DATA_BLOCK "DB_Alarms"   // DB44
{ S7_Optimized_Access := 'FALSE' }
AUTHOR : Heaten
VERSION : 0.1
// stored: AutoNumber true, DBAccessibleFromOPCUA true, DBAccessibleFromWebserver true, IsOnlyStoredInLoadMemory false, IsWriteProtectedInAS false
   VAR RETAIN
      bAckAll : Bool := FALSE;   // Global alarm acknowledge
      bCommonAlarm : Bool := FALSE;   // Global common alarm
      bCriticalAlarm : Bool := FALSE;   // Global critical alarm
      "0001_WatchdogTimeoutOB1" { S7_SetPoint := 'True'} : "stEvent";
      "0003_InitCurrentSettingsFailed" { S7_SetPoint := 'True'} : "stEvent";
      "1001_ConnectionToWinCClost" { S7_SetPoint := 'True'} : "stEvent";
      "1002_EmergencyStopActive" { S7_SetPoint := 'True'} : "stEvent";
      "1003_EmergencyStopResetFailed" { S7_SetPoint := 'True'} : "stEvent";
      "1004_HBL_PS_500_X2" { S7_SetPoint := 'True'} : "stEvent";
      "1101_HBL_SC_01_CommError" { S7_SetPoint := 'True'} : "stDigitalAlarm";
      "1102_HBL_SC_02_CommError" { S7_SetPoint := 'True'} : "stDigitalAlarm";
      "1103_HBL_SC_03_CommError" { S7_SetPoint := 'True'} : "stDigitalAlarm";
      "1110_HBL_SC_10_CommError" { S7_SetPoint := 'True'} : "stDigitalAlarm";
      "1121_HBL_SC_01_Tripped" { S7_SetPoint := 'True'} : "stDigitalAlarm";
      "1122_HBL_SC_02_Tripped" { S7_SetPoint := 'True'} : "stDigitalAlarm";
      "1123_HBL_SC_03_Tripped" { S7_SetPoint := 'True'} : "stDigitalAlarm";
      "1130_HBL_SC_10_Tripped" { S7_SetPoint := 'True'} : "stDigitalAlarm";
      "1140_HBL_SC_01_RunFailure" { S7_SetPoint := 'True'} : "stDigitalAlarm";
      "1142_HBL_SC_02_RunFailure" { S7_SetPoint := 'True'} : "stDigitalAlarm";
      "1143_HBL_SC_03_RunFailure" { S7_SetPoint := 'True'} : "stDigitalAlarm";
      "1150_HBL_SC_10_RunFailure" { S7_SetPoint := 'True'} : "stDigitalAlarm";
      "1201_HBL_PT_517_Fault" { S7_SetPoint := 'True'} : "stEvent";
      "1202_HBL_PT_612_Fault" { S7_SetPoint := 'True'} : "stEvent";
      "1203_HBL_PT_519_Fault" { S7_SetPoint := 'True'} : "stEvent";
      "1204_HBL_PT_544_Fault" { S7_SetPoint := 'True'} : "stEvent";
      "1205_HBL_TT_516_Fault" { S7_SetPoint := 'True'} : "stEvent";
      "1206_HBL_TT_611_Fault" { S7_SetPoint := 'True'} : "stEvent";
      "1207_HBL_TT_901_Fault" { S7_SetPoint := 'True'} : "stEvent";
      "1208_HBL_TT_518_Fault" { S7_SetPoint := 'True'} : "stEvent";
      "1209_HBL_HCV_576_A1_Fault" { S7_SetPoint := 'True'} : "stEvent";
      "1210_HBL_TT_573_Fault" { S7_SetPoint := 'True'} : "stEvent";
      "1212_HBL_TT_543_Fault" { S7_SetPoint := 'True'} : "stEvent";
      "1213_HBL_TT_546_Fault" { S7_SetPoint := 'True'} : "stEvent";
      "1214_HBL_TT_542_Fault" { S7_SetPoint := 'True'} : "stEvent";
      "1215_HBL_TT_571_Fault" { S7_SetPoint := 'True'} : "stEvent";
      "1216_HBL_TT_16_Fault" { S7_SetPoint := 'True'} : "stEvent";
      "1217_HBL_TT_17_Fault" { S7_SetPoint := 'True'} : "stEvent";
      "1218_HBL_TT_18_Fault" { S7_SetPoint := 'True'} : "stEvent";
      "1220_HBL_PT_960_Fault" { S7_SetPoint := 'True'} : "stEvent";
      "1221_HBL_PT_05_Fault" { S7_SetPoint := 'True'} : "stEvent";
      "1223_HBL_TT_03_Fault" { S7_SetPoint := 'True'} : "stEvent";
      "1224_HBL_TT_23_Fault" { S7_SetPoint := 'True'} : "stEvent";
      "1225_HBL_TT_24_Fault" { S7_SetPoint := 'True'} : "stEvent";
      "1226_HBL_TT_25_Fault" { S7_SetPoint := 'True'} : "stEvent";
      "1227_HBL_LT_610_Fault" { S7_SetPoint := 'True'} : "stEvent";
      "1228_HBL_TT_21_Fault" { S7_SetPoint := 'True'} : "stEvent";
      "1229_HBL_TT_22_Fault" { S7_SetPoint := 'True'} : "stEvent";
      "1230_HBL_LT_02_Fault" { S7_SetPoint := 'True'} : "stEvent";   // Deprecated
      "1231_HBL_HCV_578_A1_Fault" { S7_SetPoint := 'True'} : "stEvent";
      "1232_HBL_PT_503_Fault" { S7_SetPoint := 'True'} : "stEvent";
      "1233_HBL_TT_20_Fault" { S7_SetPoint := 'True'} : "stDigitalAlarm";
      "1234_HBL_PT_14_Fault" { S7_SetPoint := 'True'} : "stEvent";   // Deprecated
      "1235_HBL_PT_18_Fault" { S7_SetPoint := 'True'} : "stEvent";   // Deprecated
      "1236_HBL_PT_19_Fault" { S7_SetPoint := 'True'} : "stEvent";   // Deprecated
      "1237_HBL_PT_25_Fault" { S7_SetPoint := 'True'} : "stEvent";   // Deprecated
      "1238_HBL_TT_31_Fault" { S7_SetPoint := 'True'} : "stEvent";   // Deprecated
      "1239_HBL_TT_33_Fault" { S7_SetPoint := 'True'} : "stEvent";   // Deprecated
      "1240_HBL_TT_35_Fault" { S7_SetPoint := 'True'} : "stEvent";   // Deprecated
      "1241_HBL_HCV_576_Fault" { S7_SetPoint := 'True'} : "stEvent";
      "1242_HBL_HCV_578_Fault" { S7_SetPoint := 'True'} : "stEvent";
      "1243_HBL_PT_902_Fault" { S7_SetPoint := 'True'} : "stEvent";
      "1244_HBL_PT_572_Fault" { S7_SetPoint := 'True'} : "stEvent";
      "1245_HBL_PT_09_Fault" { S7_SetPoint := 'True'} : "stEvent";   // Deprecated
      "1246_HBL_PT_547_Fault" { S7_SetPoint := 'True'} : "stEvent";
      "1247_HBL_PT_541_Fault" { S7_SetPoint := 'True'} : "stEvent";
      "1248_HBL_PT_531_Fault" { S7_SetPoint := 'True'} : "stEvent";
      "1249_HBL_PT_701_Fault" { S7_SetPoint := 'True'} : "stEvent";
      "1251_HBL_PT_534_Fault" { S7_SetPoint := 'True'} : "stEvent";
      "1252_HBL_TT_540_Fault" { S7_SetPoint := 'True'} : "stEvent";
      "1253_HBL_TT_530_Fault" { S7_SetPoint := 'True'} : "stEvent";
      "1254_HBL_TT_533_Fault" { S7_SetPoint := 'True'} : "stEvent";
      "1255_HBL_CT_01_Fault" { S7_SetPoint := 'True'} : "stEvent";
      "1256_HBL_CT_615_Fault" { S7_SetPoint := 'True'} : "stEvent";
      "1257_HBL_CT_03_Fault" { S7_SetPoint := 'True'} : "stEvent";
      "1258_HBL_TT_26_Fault" { S7_SetPoint := 'True'} : "stEvent";
      "1259_HBL_TT_27_Fault" { S7_SetPoint := 'True'} : "stEvent";
      "1260_HBL_FT_520_Fault" { S7_SetPoint := 'True'} : "stEvent";
      "1262_HBL_TT_504_Fault" { S7_SetPoint := 'True'} : "stEvent";
      "1263_HBL_TT_34_Fault" { S7_SetPoint := 'True'} : "stEvent";
      "1264_HBL_PT_961_Fault" { S7_SetPoint := 'True'} : "stEvent";
      "1265_HBL_TT_502_Fault" { S7_SetPoint := 'True'} : "stEvent";
      "1266_HBL_LT_510_Fault" { S7_SetPoint := 'True'} : "stEvent";
      "1267_HBL_PT_511_Fault" { S7_SetPoint := 'True'} : "stEvent";
      "1268_HBL_TT_512_Fault" { S7_SetPoint := 'True'} : "stEvent";
      "1269_HBL_TT_532_Fault" { S7_SetPoint := 'True'} : "stEvent";
      "1270_HBL_AT_535_Fault" { S7_SetPoint := 'True'} : "stEvent";
      "1271_HBL_AT_545_Fault" { S7_SetPoint := 'True'} : "stEvent";
      "1272_HBL_PT_635_Fault" { S7_SetPoint := 'True'} : "stEvent";
      "1273_HBL_PT_636_Fault" { S7_SetPoint := 'True'} : "stEvent";
      "1274_HBL_LT_650_Fault" { S7_SetPoint := 'True'} : "stEvent";
      "1275_HBL_PT_651_Fault" { S7_SetPoint := 'True'} : "stEvent";
      "1276_HBL_PT_702_Fault" { S7_SetPoint := 'True'} : "stEvent";
      "1277_HBL_HCV_514_Fault" { S7_SetPoint := 'True'} : "stEvent";
      "1278_HBL_HCV_514_A1_Fault" { S7_SetPoint := 'True'} : "stEvent";
      "1279_HBL_HCV_515_Fault" { S7_SetPoint := 'True'} : "stEvent";
      "1280_HBL_HCV_515_A1_Fault" { S7_SetPoint := 'True'} : "stEvent";
      "1281_HBL_HCV_548_Fault" { S7_SetPoint := 'True'} : "stEvent";
      "1282_HBL_HCV_548_A1_Fault" { S7_SetPoint := 'True'} : "stEvent";
      "1283_HBL_HCV_575_Fault" { S7_SetPoint := 'True'} : "stEvent";
      "1284_HBL_HCV_575_A1_Fault" { S7_SetPoint := 'True'} : "stEvent";
      "1285_HBL_HCV_577_Fault" { S7_SetPoint := 'True'} : "stEvent";
      "1286_HBL_HCV_577_A1_Fault" { S7_SetPoint := 'True'} : "stEvent";
      "1287_HBL_HCV_579_Fault" { S7_SetPoint := 'True'} : "stEvent";
      "1288_HBL_HCV_579_A1_Fault" { S7_SetPoint := 'True'} : "stEvent";
      "1289_HBL_HCV_616_Fault" { S7_SetPoint := 'True'} : "stEvent";
      "1290_HBL_HCV_616_A1_Fault" { S7_SetPoint := 'True'} : "stEvent";
      "1291_HBL_HCV_700_Fault" { S7_SetPoint := 'True'} : "stEvent";
      "1292_HBL_HCV_700_A1_Fault" { S7_SetPoint := 'True'} : "stEvent";
      "1293_HBL_PT_618_Fault" { S7_SetPoint := 'True'} : "stEvent";
      "1294_HBL_LS_632_Fault" { S7_SetPoint := 'True'} : "stDigitalAlarm";
      "1295_HBL_LS_633_Fault" { S7_SetPoint := 'True'} : "stDigitalAlarm";
      "2018_HBL_PT_05_High" { S7_SetPoint := 'True'} : "stLimitAlarm";
      "2028_HBL_PT_17_Low" { S7_SetPoint := 'True'} : "stLimitAlarm";
      "2058_HBL_TT_03_Low" { S7_SetPoint := 'True'} : "stLimitAlarm";
      "2100_HBL_TT_03_High" { S7_SetPoint := 'True'} : "stLimitAlarm";
      "2101_HBL_TT_901_High" { S7_SetPoint := 'True'} : "stLimitAlarm";
      "2102_HBL_PT_503_High" { S7_SetPoint := 'True'} : "stLimitAlarm";
      "2103_HBL_TT_518_High" { S7_SetPoint := 'True'} : "stLimitAlarm";
      "2105_HBL_TT_546_High" { S7_SetPoint := 'True'} : "stLimitAlarm";
      "2106_HBL_TT_17_High" { S7_SetPoint := 'True'} : "stLimitAlarm";
      "2107_HBL_TT_16_High" { S7_SetPoint := 'True'} : "stLimitAlarm";
      "2108_HBL_TT_18_High" { S7_SetPoint := 'True'} : "stLimitAlarm";
      "2109_HBL_TT_20_High" { S7_SetPoint := 'True'} : "stLimitAlarm";
      "2110_HBL_TT_21_High" { S7_SetPoint := 'True'} : "stLimitAlarm";
      "2111_HBL_TT_22_High" { S7_SetPoint := 'True'} : "stLimitAlarm";
      "2112_HBL_LT_02_High" { S7_SetPoint := 'True'} : "stLimitAlarm";   // Deprecated
      "2113_HBL_CT_01_High" { S7_SetPoint := 'True'} : "stLimitAlarm";
      "2114_HBL_CT_615_High" { S7_SetPoint := 'True'} : "stLimitAlarm";
      "2115_HBL_PT_17_LowLow" { S7_SetPoint := 'True'} : "stLimitAlarm";
      "2116_HBL_PT_503_HighHigh" { S7_SetPoint := 'True'} : "stLimitAlarm";
      "2117_HBL_TT_542_Low" { S7_SetPoint := 'True'} : "stLimitAlarm";
      "2301_HeatSourceTempDropCritical" { S7_SetPoint := 'True'} : "stLimitAlarm";
      "2302_HeatSourceTempRiseCritical" { S7_SetPoint := 'True'} : "stLimitAlarm";
      "2303_SuperheatCompressor_High" { S7_SetPoint := 'True'} : "stLimitAlarm";
      "2304_SuperheatCompressor_Low" { S7_SetPoint := 'True'} : "stLimitAlarm";
      "2305_OilFilterDeltaP_High" { S7_SetPoint := 'True'} : "stLimitAlarm";
      "2306_OilFilterDeltaP_HighHigh" { S7_SetPoint := 'True'} : "stLimitAlarm";
      "2307_EvaporatorDischargePressureMeanValue" { S7_SetPoint := 'True'} : "stEvent";
      "2308_EvaporatorDischargePressureHigh" { S7_SetPoint := 'True'} : "stLimitAlarm";
      "2309_OilSeparatorStage1High" { S7_SetPoint := 'True'} : "stDigitalAlarm";
      "3020_SuperheatControlRegulatorFault" { S7_SetPoint := 'True'} : "stEvent";
      "3030_PinchControlRegulatorfault" { S7_SetPoint := 'True'} : "stEvent";
      "3400_HydrolockProtectionActive" { S7_SetPoint := 'True'} : "stEvent";
      "3401_DripPanLevelHigh" { S7_SetPoint := 'True'} : "stDigitalAlarm";
      "5000_OilHeatingActivationFailure" { S7_SetPoint := 'True'} : "stDigitalAlarm";
      "5001_OilHeatingDeactivationFailure" { S7_SetPoint := 'True'} : "stDigitalAlarm";
      "5200_CPC_LT_870_Fault" { S7_SetPoint := 'True'} : "stEvent";
      "5201_CPC_TT_871_Fault" { S7_SetPoint := 'True'} : "stEvent";
      "5202_CPC_PT_872_Fault" { S7_SetPoint := 'True'} : "stEvent";
      "5203_CPC_SC_01_CommError" { S7_SetPoint := 'True'} : "stDigitalAlarm";   // Deprecated
      "5204_CPC_SC_01_Tripped" { S7_SetPoint := 'True'} : "stDigitalAlarm";   // Deprecated
      "5205_CPC_LT_870_High" { S7_SetPoint := 'True'} : "stLimitAlarm";
      "5206_CPC_PT_862_Fault" { S7_SetPoint := 'True'} : "stEvent";
      "5250_SSC_TT_01_Fault" { S7_SetPoint := 'True'} : "stEvent";
      "5251_SSC_TT_02_Fault" { S7_SetPoint := 'True'} : "stEvent";
      "5252_SSC_TT_03_Fault" { S7_SetPoint := 'True'} : "stEvent";
      "5253_SSC_TT_04_Fault" { S7_SetPoint := 'True'} : "stEvent";
      "5254_SSC_PIT_01_Fault" { S7_SetPoint := 'True'} : "stEvent";
      "5255_SSC_PDT_01_Fault" { S7_SetPoint := 'True'} : "stEvent";
      "5256_SSC_LT_01_Fault" { S7_SetPoint := 'True'} : "stEvent";
      "5257_SSC_LT_01_Low" { S7_SetPoint := 'True'} : "stLimitAlarm";
      "5258_SSC_PDT_01_High" { S7_SetPoint := 'True'} : "stLimitAlarm";
      "5259_SSC_TT_02_High" { S7_SetPoint := 'True'} : "stLimitAlarm";
      "5260_SSC_TT_03_Low" { S7_SetPoint := 'True'} : "stLimitAlarm";
      "5261_SSC_PIT_01_Low" { S7_SetPoint := 'True'} : "stLimitAlarm";
      "5262_DeltaT_ShaftSealHigh" { S7_SetPoint := 'True'} : "stLimitAlarm";
      "5263_SSC_PIT_01_High" { S7_SetPoint := 'True'} : "stLimitAlarm";
      "5268_ShaftSealSystemShutdown" { S7_SetPoint := 'True'} : "stDigitalAlarm";
      "9023_HBL_HCV_576_Deviation" { S7_SetPoint := 'True'} : "stDeviationAlarm";
      "9024_HBL_HCV_578_Deviation" { S7_SetPoint := 'True'} : "stDeviationAlarm";
      "9025_HBL_HCV_577_Deviation" { S7_SetPoint := 'True'} : "stDeviationAlarm";
      "9026_HBL_HCV_579_Deviation" { S7_SetPoint := 'True'} : "stDeviationAlarm";
      "9027_HBL_HCV_575_Deviation" { S7_SetPoint := 'True'} : "stDeviationAlarm";
      "9028_HBL_HCV_616_Deviation" { S7_SetPoint := 'True'} : "stDeviationAlarm";
      "9029_HBL_HCV_700_Deviation" { S7_SetPoint := 'True'} : "stDeviationAlarm";
      "9030_HBL_HCV_514_Deviation" { S7_SetPoint := 'True'} : "stDeviationAlarm";
      "9031_HBL_HCV_548_Deviation" { S7_SetPoint := 'True'} : "stDeviationAlarm";
   END_VAR
BEGIN
   "0001_WatchdogTimeoutOB1".bEnable := true;
   "0003_InitCurrentSettingsFailed".bEnable := TRUE;
   "1001_ConnectionToWinCClost".bEnable := TRUE;
   "1002_EmergencyStopActive".bEnable := TRUE;
   "1003_EmergencyStopResetFailed".bEnable := TRUE;
   "1101_HBL_SC_01_CommError".bEnable := true;
   "1101_HBL_SC_01_CommError".bInput := FALSE;
   "1101_HBL_SC_01_CommError".tActivationDelay := T#1S;
   "1102_HBL_SC_02_CommError".bEnable := true;
   "1102_HBL_SC_02_CommError".tActivationDelay := T#1s;
   "1103_HBL_SC_03_CommError".bEnable := true;
   "1103_HBL_SC_03_CommError".tActivationDelay := T#1s;
   "1110_HBL_SC_10_CommError".bEnable := TRUE;
   "1110_HBL_SC_10_CommError".bInput := FALSE;
   "1110_HBL_SC_10_CommError".tActivationDelay := T#5s;
   "1121_HBL_SC_01_Tripped".bEnable := TRUE;
   "1121_HBL_SC_01_Tripped".bInput := FALSE;
   "1121_HBL_SC_01_Tripped".tActivationDelay := T#0MS;
   "1122_HBL_SC_02_Tripped".bEnable := true;
   "1122_HBL_SC_02_Tripped".tActivationDelay := T#0s;
   "1123_HBL_SC_03_Tripped".bEnable := true;
   "1130_HBL_SC_10_Tripped".bEnable := TRUE;
   "1130_HBL_SC_10_Tripped".bInput := FALSE;
   "1130_HBL_SC_10_Tripped".tActivationDelay := T#3s;
   "1140_HBL_SC_01_RunFailure".bEnable := TRUE;
   "1140_HBL_SC_01_RunFailure".bInput := FALSE;
   "1140_HBL_SC_01_RunFailure".tActivationDelay := T#0MS;
   "1142_HBL_SC_02_RunFailure".bEnable := true;
   "1142_HBL_SC_02_RunFailure".tActivationDelay := T#3s;
   "1143_HBL_SC_03_RunFailure".bEnable := true;
   "1143_HBL_SC_03_RunFailure".tActivationDelay := T#3s;
   "1150_HBL_SC_10_RunFailure".bEnable := TRUE;
   "1150_HBL_SC_10_RunFailure".bInput := FALSE;
   "1150_HBL_SC_10_RunFailure".tActivationDelay := T#3s;
   "1201_HBL_PT_517_Fault".bEnable := true;
   "1202_HBL_PT_612_Fault".bEnable := true;
   "1203_HBL_PT_519_Fault".bEnable := true;
   "1204_HBL_PT_544_Fault".bEnable := true;
   "1205_HBL_TT_516_Fault".bEnable := true;
   "1206_HBL_TT_611_Fault".bEnable := true;
   "1207_HBL_TT_901_Fault".bEnable := true;
   "1208_HBL_TT_518_Fault".bEnable := true;
   "1209_HBL_HCV_576_A1_Fault".bEnable := true;
   "1210_HBL_TT_573_Fault".bEnable := true;
   "1212_HBL_TT_543_Fault".bEnable := true;
   "1213_HBL_TT_546_Fault".bEnable := true;
   "1214_HBL_TT_542_Fault".bEnable := true;
   "1215_HBL_TT_571_Fault".bEnable := true;
   "1216_HBL_TT_16_Fault".bEnable := true;
   "1217_HBL_TT_17_Fault".bEnable := true;
   "1218_HBL_TT_18_Fault".bEnable := true;
   "1220_HBL_PT_960_Fault".bEnable := true;
   "1221_HBL_PT_05_Fault".bEnable := true;
   "1223_HBL_TT_03_Fault".bEnable := true;
   "1224_HBL_TT_23_Fault".bEnable := true;
   "1225_HBL_TT_24_Fault".bEnable := true;
   "1226_HBL_TT_25_Fault".bEnable := true;
   "1227_HBL_LT_610_Fault".bEnable := true;
   "1228_HBL_TT_21_Fault".bEnable := true;
   "1229_HBL_TT_22_Fault".bEnable := true;
   "1230_HBL_LT_02_Fault".bEnable := false;
   "1231_HBL_HCV_578_A1_Fault".bEnable := true;
   "1232_HBL_PT_503_Fault".bEnable := true;
   "1233_HBL_TT_20_Fault".bEnable := TRUE;
   "1233_HBL_TT_20_Fault".tActivationDelay := T#5S;
   "1234_HBL_PT_14_Fault".bEnable := true;
   "1235_HBL_PT_18_Fault".bEnable := true;
   "1236_HBL_PT_19_Fault".bEnable := true;
   "1237_HBL_PT_25_Fault".bEnable := false;
   "1238_HBL_TT_31_Fault".bEnable := true;
   "1239_HBL_TT_33_Fault".bEnable := true;
   "1240_HBL_TT_35_Fault".bEnable := true;
   "1241_HBL_HCV_576_Fault".bEnable := true;
   "1242_HBL_HCV_578_Fault".bEnable := true;
   "1243_HBL_PT_902_Fault".bEnable := true;
   "1244_HBL_PT_572_Fault".bEnable := true;
   "1245_HBL_PT_09_Fault".bEnable := true;
   "1246_HBL_PT_547_Fault".bEnable := true;
   "1247_HBL_PT_541_Fault".bEnable := true;
   "1248_HBL_PT_531_Fault".bEnable := true;
   "1249_HBL_PT_701_Fault".bEnable := true;
   "1251_HBL_PT_534_Fault".bEnable := true;
   "1252_HBL_TT_540_Fault".bEnable := true;
   "1253_HBL_TT_530_Fault".bEnable := true;
   "1254_HBL_TT_533_Fault".bEnable := true;
   "1255_HBL_CT_01_Fault".bEnable := true;
   "1256_HBL_CT_615_Fault".bEnable := true;
   "1258_HBL_TT_26_Fault".bEnable := true;
   "1259_HBL_TT_27_Fault".bEnable := true;
   "1260_HBL_FT_520_Fault".bEnable := true;
   "1262_HBL_TT_504_Fault".bEnable := true;
   "1263_HBL_TT_34_Fault".bEnable := true;
   "1264_HBL_PT_961_Fault".bEnable := true;
   "1265_HBL_TT_502_Fault".bEnable := true;
   "1266_HBL_LT_510_Fault".bEnable := true;
   "1267_HBL_PT_511_Fault".bEnable := true;
   "1268_HBL_TT_512_Fault".bEnable := true;
   "1269_HBL_TT_532_Fault".bEnable := true;
   "1270_HBL_AT_535_Fault".bEnable := true;
   "1271_HBL_AT_545_Fault".bEnable := true;
   "1272_HBL_PT_635_Fault".bEnable := true;
   "1273_HBL_PT_636_Fault".bEnable := true;
   "1274_HBL_LT_650_Fault".bEnable := true;
   "1275_HBL_PT_651_Fault".bEnable := true;
   "1276_HBL_PT_702_Fault".bEnable := true;
   "1283_HBL_HCV_575_Fault".bEnable := true;
   "1284_HBL_HCV_575_A1_Fault".bEnable := true;
   "1285_HBL_HCV_577_Fault".bEnable := true;
   "1286_HBL_HCV_577_A1_Fault".bEnable := true;
   "1287_HBL_HCV_579_Fault".bEnable := true;
   "1288_HBL_HCV_579_A1_Fault".bEnable := true;
   "1289_HBL_HCV_616_Fault".bEnable := true;
   "1290_HBL_HCV_616_A1_Fault".bEnable := true;
   "1291_HBL_HCV_700_Fault".bEnable := true;
   "1292_HBL_HCV_700_A1_Fault".bEnable := true;
   "1293_HBL_PT_618_Fault".bEnable := true;
   "1294_HBL_LS_632_Fault".tActivationDelay := t#5S;
   "2018_HBL_PT_05_High".bEnable := true;
   "2018_HBL_PT_05_High".fLimit := 1600.0;
   "2018_HBL_PT_05_High".fHysteresis := 0.0;
   "2018_HBL_PT_05_High".tActivationDelay := T#0MS;
   "2028_HBL_PT_17_Low".bEnable := true;
   "2028_HBL_PT_17_Low".fLimit := 30.0;
   "2028_HBL_PT_17_Low".fHysteresis := 0.0;
   "2028_HBL_PT_17_Low".tActivationDelay := T#30s;
   "2058_HBL_TT_03_Low".bEnable := true;
   "2058_HBL_TT_03_Low".fLimit := 0.0;
   "2058_HBL_TT_03_Low".fHysteresis := 1.0;
   "2058_HBL_TT_03_Low".tActivationDelay := T#180s;
   "2100_HBL_TT_03_High".bEnable := true;
   "2100_HBL_TT_03_High".tActivationDelay := T#0MS;
   "2101_HBL_TT_901_High".bEnable := true;
   "2101_HBL_TT_901_High".fHysteresis := 5.0;
   "2101_HBL_TT_901_High".tActivationDelay := T#5s;
   "2102_HBL_PT_503_High".bEnable := true;
   "2102_HBL_PT_503_High".tActivationDelay := T#1s;
   "2103_HBL_TT_518_High".bEnable := true;
   "2103_HBL_TT_518_High".tActivationDelay := T#1s;
   "2105_HBL_TT_546_High".bEnable := true;
   "2106_HBL_TT_17_High".bEnable := true;
   "2106_HBL_TT_17_High".tActivationDelay := T#10s;
   "2107_HBL_TT_16_High".bEnable := true;
   "2107_HBL_TT_16_High".tActivationDelay := T#10s;
   "2108_HBL_TT_18_High".bEnable := true;
   "2108_HBL_TT_18_High".tActivationDelay := T#10s;
   "2109_HBL_TT_20_High".bEnable := true;
   "2109_HBL_TT_20_High".tActivationDelay := T#0s;
   "2110_HBL_TT_21_High".bEnable := true;
   "2110_HBL_TT_21_High".fHysteresis := 5.0;
   "2110_HBL_TT_21_High".tActivationDelay := T#10s;
   "2111_HBL_TT_22_High".bEnable := true;
   "2111_HBL_TT_22_High".fHysteresis := 5.0;
   "2111_HBL_TT_22_High".tActivationDelay := T#10s;
   "2112_HBL_LT_02_High".bEnable := true;
   "2112_HBL_LT_02_High".tActivationDelay := T#5s;
   "2113_HBL_CT_01_High".bEnable := true;
   "2113_HBL_CT_01_High".fHysteresis := 50.0;
   "2114_HBL_CT_615_High".bEnable := true;
   "2114_HBL_CT_615_High".fHysteresis := 50.0;
   "2115_HBL_PT_17_LowLow".bEnable := true;
   // "2115_HBL_PT_17_LowLow".fLimit : Dynamic threshold!!
   "2115_HBL_PT_17_LowLow".tActivationDelay := T#2s;
   "2116_HBL_PT_503_HighHigh".bEnable := true;
   "2117_HBL_TT_542_Low".bEnable := true;
   "2117_HBL_TT_542_Low".fLimit := 5.0;
   "2117_HBL_TT_542_Low".fHysteresis := 1.0;
   "2117_HBL_TT_542_Low".tActivationDelay := T#2s;
   "2301_HeatSourceTempDropCritical".bEnable := true;
   "2302_HeatSourceTempRiseCritical".bEnable := true;
   "2303_SuperheatCompressor_High".bEnable := true;
   "2304_SuperheatCompressor_Low".bEnable := true;
   "2305_OilFilterDeltaP_High".bEnable := true;
   "2305_OilFilterDeltaP_High".fLimit := 30.0;
   "2305_OilFilterDeltaP_High".fHysteresis := 2.0;
   "2305_OilFilterDeltaP_High".tActivationDelay := T#10s;
   "2306_OilFilterDeltaP_HighHigh".bEnable := true;
   "2306_OilFilterDeltaP_HighHigh".fLimit := 100.0;
   "2306_OilFilterDeltaP_HighHigh".fHysteresis := 5.0;
   "2306_OilFilterDeltaP_HighHigh".tActivationDelay := T#5s;
   "2307_EvaporatorDischargePressureMeanValue".bEnable := true;
   "2308_EvaporatorDischargePressureHigh".bEnable := true;
   "2309_OilSeparatorStage1High".tActivationDelay := T#5m;
   "3020_SuperheatControlRegulatorFault".bEnable := true;
   "3400_HydrolockProtectionActive".bEnable := TRUE;
   "3401_DripPanLevelHigh".bEnable := false;
   "3401_DripPanLevelHigh".tActivationDelay := T#3S;
   "5000_OilHeatingActivationFailure".bEnable := TRUE;
   "5000_OilHeatingActivationFailure".bInput := FALSE;
   "5000_OilHeatingActivationFailure".tActivationDelay := T#2s;
   "5001_OilHeatingDeactivationFailure".bEnable := TRUE;
   "5001_OilHeatingDeactivationFailure".bInput := FALSE;
   "5001_OilHeatingDeactivationFailure".tActivationDelay := T#2s;
   "5200_CPC_LT_870_Fault".bEnable := true;
   "5201_CPC_TT_871_Fault".bEnable := true;
   "5202_CPC_PT_872_Fault".bEnable := true;
   "5203_CPC_SC_01_CommError".bEnable := false;
   "5203_CPC_SC_01_CommError".tActivationDelay := T#1S;
   "5204_CPC_SC_01_Tripped".bEnable := false;
   "5204_CPC_SC_01_Tripped".tActivationDelay := T#0MS;
   "5205_CPC_LT_870_High".bEnable := true;
   "5205_CPC_LT_870_High".fHysteresis := 2.0;
   "5205_CPC_LT_870_High".tActivationDelay := T#2S;
   "5206_CPC_PT_862_Fault".bEnable := true;
   "5250_SSC_TT_01_Fault".bEnable := true;
   "5251_SSC_TT_02_Fault".bEnable := true;
   "5252_SSC_TT_03_Fault".bEnable := true;
   "5253_SSC_TT_04_Fault".bEnable := true;
   "5254_SSC_PIT_01_Fault".bEnable := true;
   "5255_SSC_PDT_01_Fault".bEnable := true;
   "5256_SSC_LT_01_Fault".bEnable := true;
   "5257_SSC_LT_01_Low".bEnable := true;
   "5257_SSC_LT_01_Low".fLimit := 5.0;
   "5257_SSC_LT_01_Low".fHysteresis := 2.0;
   "5257_SSC_LT_01_Low".tActivationDelay := T#2S;
   "5258_SSC_PDT_01_High".bEnable := true;
   "5258_SSC_PDT_01_High".fLimit := 200.0;
   "5258_SSC_PDT_01_High".fHysteresis := 10.0;
   "5258_SSC_PDT_01_High".tActivationDelay := T#5S;
   "5259_SSC_TT_02_High".bEnable := true;
   "5259_SSC_TT_02_High".fLimit := 110.0;
   "5259_SSC_TT_02_High".fHysteresis := 2.0;
   "5259_SSC_TT_02_High".tActivationDelay := T#5S;
   "5260_SSC_TT_03_Low".bEnable := true;
   "5260_SSC_TT_03_Low".fLimit := 10.0;
   "5260_SSC_TT_03_Low".fHysteresis := 0.5;
   "5260_SSC_TT_03_Low".tActivationDelay := T#5S;
   "5261_SSC_PIT_01_Low".bEnable := true;
   "5261_SSC_PIT_01_Low".fLimit := 840.0;
   "5261_SSC_PIT_01_Low".fHysteresis := 10.0;
   "5261_SSC_PIT_01_Low".tActivationDelay := T#2S;
   "5262_DeltaT_ShaftSealHigh".bEnable := true;
   "5262_DeltaT_ShaftSealHigh".fLimit := 11.0;
   "5262_DeltaT_ShaftSealHigh".fHysteresis := 0.5;
   "5262_DeltaT_ShaftSealHigh".tActivationDelay := T#30S;
   "5263_SSC_PIT_01_High".bEnable := true;
   "5263_SSC_PIT_01_High".fLimit := 1400.0;
   "5263_SSC_PIT_01_High".fHysteresis := 5.0;
   "5263_SSC_PIT_01_High".tActivationDelay := T#2S;
   "5268_ShaftSealSystemShutdown".bEnable := false;
   "9023_HBL_HCV_576_Deviation".bEnable := true;
   "9023_HBL_HCV_576_Deviation".fDeviationLimit := 4.0;   // [%]
   "9023_HBL_HCV_576_Deviation".tActivationDelay := T#30s;
   "9024_HBL_HCV_578_Deviation".bEnable := true;
   "9024_HBL_HCV_578_Deviation".fDeviationLimit := 4.0;   // [%]
   "9024_HBL_HCV_578_Deviation".tActivationDelay := T#30s;
   "9025_HBL_HCV_577_Deviation".bEnable := true;
   "9025_HBL_HCV_577_Deviation".fDeviationLimit := 4.0;
   "9025_HBL_HCV_577_Deviation".tActivationDelay := T#30s;
   "9026_HBL_HCV_579_Deviation".bEnable := true;
   "9026_HBL_HCV_579_Deviation".fDeviationLimit := 4.0;
   "9026_HBL_HCV_579_Deviation".tActivationDelay := T#30s;
   "9027_HBL_HCV_575_Deviation".bEnable := true;
   "9027_HBL_HCV_575_Deviation".fDeviationLimit := 4.0;
   "9027_HBL_HCV_575_Deviation".tActivationDelay := T#5s;
   "9028_HBL_HCV_616_Deviation".bEnable := true;
   "9028_HBL_HCV_616_Deviation".fDeviationLimit := 4.0;
   "9028_HBL_HCV_616_Deviation".tActivationDelay := T#5s;
   "9029_HBL_HCV_700_Deviation".bEnable := true;
   "9029_HBL_HCV_700_Deviation".fDeviationLimit := 4.0;
   "9029_HBL_HCV_700_Deviation".tActivationDelay := T#5s;
   "9030_HBL_HCV_514_Deviation".bEnable := true;
   "9030_HBL_HCV_514_Deviation".fDeviationLimit := 4.0;
   "9030_HBL_HCV_514_Deviation".tActivationDelay := T#5s;
   "9031_HBL_HCV_548_Deviation".bEnable := true;
   "9031_HBL_HCV_548_Deviation".fDeviationLimit := 4.0;
   "9031_HBL_HCV_548_Deviation".tActivationDelay := T#5s;
END_DATA_BLOCK

DATA_BLOCK "DB_Application"   // DB9
{ S7_Optimized_Access := 'FALSE' }
VERSION : 0.1
// stored: AutoNumber true, DBAccessibleFromOPCUA true, DBAccessibleFromWebserver true, IsOnlyStoredInLoadMemory false, IsWriteProtectedInAS false
   VAR
      ToHB : Struct
         StartRequest : Bool;
         StopRequest : Bool;
         AlarmAcknowledge : Bool;
         EmergencyStopResetRequest : Bool;
         FastStopRequest : Bool;
         HydrolockProtection : Bool;
         SpareCommand6 : Bool;
         SpareCommand7 : Bool;
         SuperheatManualMode : Bool;
         HeatSinkOutManualMode : Bool;
         PerformanceControlManualMode : Bool;
         OilHeatingRegulatorManualMode : Bool;
         ExpansionValveRegulatorManualMode : Bool;
         PinchRegulatorManualMode : Bool;
         SpareManualMode6 : Bool;
         SpareManualMode7 : Bool;
         PumaCommOk : Bool;   // 1 = communication OK, 0 = communication dead
         HeatSourceOk : Bool;   // 1 = Source ready, 0 = source not ready
         HeatSinkOk : Bool;   // 1 = Sink ready, 0 = sink not ready
         SpareGroup2Command3 : Bool;
         SpareGroup2Command4 : Bool;
         SpareGroup2Command5 : Bool;
         SpareGroup2Command6 : Bool;
         SpareGroup2Command7 : Bool;
         SpareGroup3Command0 : Bool;
         SpareGroup3Command1 : Bool;
         SpareGroup3Command2 : Bool;
         SpareGroup3Command3 : Bool;
         SpareGroup3Command4 : Bool;
         SpareGroup3Command5 : Bool;
         SpareGroup3Command6 : Bool;
         SpareGroup3Command7 : Bool;
         SuperheatManualValue : Real;
         HeatSinkOutManualValue : Real;
         PerformanceControlManualValue : Real;
         OilHeatingManualValue : Real;
         ExpansionValveManualValue : Real;
         PinchManualValue : Real;
         HeatboosterSetpoint : Real;
         RegulationTarget : Int;
         LivenessCounter : UInt;
         HBL_HCV_514_A1 : Real;   // If externally controlled
         HBL_HCV_548_A1 : Real;   // If externally controlled
         HBL_TT_546 : Real;   // If externally controlled
         HBL_PT_547 : Real;   // If externally controlled
         HBL_HCV_515_A1 : Real;   // If externally controlled
         HBL_TT_901 : Real;   // If externally controlled
         HBL_PT_902 : Real;   // If externally controlled
         HBL_TT_512 : Real;   // If externally controlled
         HBL_PT_511 : Real;   // If externally controlled
         HBL_PT_519 : Real;   // If externally controlled
         HBL_TT_518 : Real;   // If externally controlled
      END_STRUCT;
      FromHB : Struct
         EmergencyStop : Bool;
         OilHeatersGroup1 : Bool;
         OilHeatersGroup2 : Bool;
         HBL_SC_01_Ready : Bool;
         HBL_SC_01_Run : Bool;
         HBL_SC_01_Tripped : Bool;
         HBL_SC_02_Ready : Bool;
         HBL_SC_02_Run : Bool;
         HBL_SC_02_Tripped : Bool;
         HBL_SC_10_Ready : Bool;
         HBL_SC_10_Run : Bool;
         HBL_SC_10_Tripped : Bool;
         HBL_HV_630 : Bool;
         HBL_HV_631 : Bool;
         HBL_HV_860 : Bool;
         HBL_HV_861 : Bool;
         HBL_HV_114 : Bool;
         HBL_HV_115 : Bool;
         CPC_P_01 : Bool;
         SSC_P_01 : Bool;
         SSC_F_01 : Bool;
         SSC_P_02 : Bool;
         HBL_LS_01 : Bool;
         HBL_LS_02 : Bool;
         HBL_HV_112 : Bool;
         HBL_HV_113 : Bool;
         HBL_LSH_62 : Bool;
         HBL_LSL_63 : Bool;
         HBL_LSH_64 : Bool;
         HBL_LSL_864 : Bool;
         HBL_LS_632 : Bool;
         HBL_LS_633 : Bool;
         HBL_SC_03_Ready : Bool;
         HBL_SC_03_Run : Bool;
         HBL_SC_03_Tripped : Bool;
         HBL_HCV_514_Force : Bool;
         HBL_HCV_548_Force : Bool;
         Spare05 : Bool;
         Spare06 : Bool;
         Spare07 : Bool;
         MachineState : Int;
         CompressorType : Int;
         SystemType : Int;
         RefrigerantType : Int;
         UptimeHours : Int;
         UptimeMinutes : Int;
         UptimeSeconds : Int;
         ActiveTimeHours : Int;
         ActiveTimeMinutes : Int;
         ActiveTimeSeconds : Int;
         RunningTimeHours : Int;
         RunningTimeMinutes : Int;
         RunningTimeSeconds : Int;
         Alarms : Array[0..159] of Bool;   // Compressed alarm bits
         HeatboosterSetpoint : Real;
         RegulationTarget : Int;
         HBL_HCV_514 : Real;   // Force setpoint
         HBL_HCV_548 : Real;   // Force setpoint
         DB_AI : Struct
            HBL_TT_502 : Real;
            HBL_PT_503 : Real;
            HBL_TT_504 : Real;
            HBL_LT_510 : Real;
            HBL_PT_511 : Real;
            HBL_TT_512 : Real;
            HBL_TT_516 : Real;
            HBL_PT_517 : Real;
            HBL_TT_518 : Real;
            HBL_PT_519 : Real;
            HBL_FT_520 : Real;
            HBL_TT_530 : Real;
            HBL_PT_531 : Real;
            HBL_TT_532 : Real;
            HBL_TT_533 : Real;
            HBL_PT_534 : Real;
            HBL_AT_535 : Real;
            HBL_TT_540 : Real;
            HBL_PT_541 : Real;
            HBL_TT_542 : Real;
            HBL_TT_543 : Real;
            HBL_PT_544 : Real;
            HBL_AT_545 : Real;
            HBL_TT_546 : Real;
            HBL_PT_547 : Real;
            HBL_TT_571 : Real;
            HBL_PT_572 : Real;
            HBL_TT_573 : Real;
            HBL_LT_610 : Real;
            HBL_TT_611 : Real;
            HBL_PT_612 : Real;
            HBL_CT_615 : Real;
            HBL_PT_618 : Real;
            HBL_PT_635 : Real;
            HBL_PT_636 : Real;
            HBL_LT_650 : Real;
            HBL_PT_651 : Real;
            HBL_PT_701 : Real;
            HBL_PT_702 : Real;
            HBL_PT_703 : Real;
            CPC_LT_870 : Real;
            CPC_TT_871 : Real;
            CPC_PT_872 : Real;
            CPC_PT_862 : Real;
            HBL_TT_901 : Real;
            HBL_PT_902 : Real;
            HBL_TT_03 : Real;
            HBL_TT_16 : Real;
            HBL_TT_17 : Real;
            HBL_TT_18 : Real;
            HBL_TT_20 : Real;
            HBL_TT_21 : Real;
            HBL_TT_22 : Real;
            HBL_TT_23 : Real;
            HBL_TT_24 : Real;
            HBL_TT_25 : Real;
            HBL_TT_26 : Real;
            HBL_TT_27 : Real;
            HBL_PT_05 : Real;
            HBL_PT_06 : Real;
            HBL_PT_17 : Real;
            HBL_CT_01 : Real;
            HBL_CT_03 : Real;
            SSC_TT_01 : Real;
            SSC_TT_02 : Real;
            SSC_TT_03 : Real;
            SSC_TT_04 : Real;
            SSC_PIT_01 : Real;
            SSC_PDT_01 : Real;
            SSC_LT_01 : Real;
         END_STRUCT;
         DB_Calc : Struct
            Compressor_CrankcaseSaturationTemperature : Real;
            Compressor_CrankcaseSuperheat : Real;
            Compressor_VolumetricEfficiency : Real;
            Compressor_IsentropicEfficiency : Real;
            Compressor_Massflow : Real;
            Heatsink_DeltaT : Real;
            Heatsink_Pinch : Real;
            Heatsink_Heatrate : Real;
            Heatsink_DeltaP : Real;
            Heatsink_Massflow : Real;
            Heatsource_DeltaT : Real;
            Heatsource_Pinch : Real;
            Heatsource_Heatrate : Real;
            Heatsource_DeltaP : Real;
            Heatsource_TemperatureRateOfChange : Real;
            Heatsource_Massflow : Real;
            HighPressPart_CompressorSaturationTemperature : Real;
            HighPressPart_CompressorSuperheat : Real;
            HighPressPart_CondenserSaturationTemperature : Real;
            HighPressPart_CondenserSubcooling : Real;
            HighPressPart_ExpansionValveSubcooling : Real;
            HighPressPart_CondenserDeltaP : Real;
            LowPressPart_EvaporatorSuperheat : Real;
            LowPressPart_CompressorSuperheat : Real;
            LowPressPart_EvaporatorSaturationTemperature : Real;
            LowPressPart_CompressorSaturationTemperature : Real;
            System_Quality : Real;
            System_COP : Real;
            System_ElectricalPower : Real;
            System_TemperatureLift : Real;
            System_MotorEfficiency : Real;
            System_FMEP : Real;
            Aux_ShaftSealDeltaT : Real;
            Aux_CPCPumpDeltaP : Real;
            Misc_EvaporatorDischargePressureMean : Real;
            Misc_EvaporatorDischargeTemperatureMin : Real;
            Misc_EvaporatorDischargeTemperatureMean : Real;
            Misc_OilFilterDeltaP : Real;
         END_STRUCT;
         DB_InverterDrives : Struct
            HBL_SC_01_A1 : Real;
            HBL_SC_01_A2 : Real;
            HBL_SC_01_A3 : Real;
            HBL_SC_02_A1 : Real;
            HBL_SC_02_A2 : Real;
            HBL_SC_02_A3 : Real;
            HBL_SC_10_A1 : Real;
            HBL_SC_10_A2 : Real;
            HBL_SC_10_A3 : Real;
            HBL_SC_03_A1 : Real;
            HBL_SC_03_A2 : Real;
            HBL_SC_03_A3 : Real;
         END_STRUCT;
         DB_Valves : Struct
            HBL_HCV_576_A1 : Real;
            HBL_HCV_578_A1 : Real;
            HBL_HCV_577_A1 : Real;
            HBL_HCV_579_A1 : Real;
            HBL_HCV_515_A1 : Real;
            HBL_HCV_575_A1 : Real;
            HBL_HCV_616_A1 : Real;
            HBL_HCV_700_A1 : Real;
            HBL_HCV_514_A1 : Real;
            HBL_HCV_548_A1 : Real;
         END_STRUCT;
      END_STRUCT;
   END_VAR
BEGIN
END_DATA_BLOCK

DATA_BLOCK "DB_Calc"   // DB45
{ S7_Optimized_Access := 'FALSE' }
AUTHOR : Heaten
VERSION : 0.1
// stored: AutoNumber true, DBAccessibleFromOPCUA true, DBAccessibleFromWebserver true, IsOnlyStoredInLoadMemory false, IsWriteProtectedInAS false
   VAR RETAIN
      Compressor : Struct
         CrankcaseSaturationTemperature : "stCalcValue";   // C
         CrankcaseSuperheat { S7_SetPoint := 'True'} : "stCalcValue";
         VolumetricEfficiency { S7_SetPoint := 'True'} : "stCalcValue";   // %
         IsentropicEfficiency { S7_SetPoint := 'True'} : "stCalcValue";   // %
         Massflow { S7_SetPoint := 'True'} : "stCalcValue";   // Refrigerant massflow (kg/h)
      END_STRUCT;
      HeatSink : Struct
         DeltaT : "stCalcValue";   // C
         Pinch { S7_SetPoint := 'True'} : "stCalcValue";   // C
         HeatRate { S7_SetPoint := 'True'} : "stCalcValue";   // kW
         DeltaP { S7_SetPoint := 'True'} : "stCalcValue";   // kPa
         Massflow { S7_SetPoint := 'True'} : "stCalcValue";   // Cooling media massflow (t/h)
      END_STRUCT;
      HeatSource : Struct
         DeltaT : "stCalcValue";   // C
         Pinch { S7_SetPoint := 'True'} : "stCalcValue";   // C
         HeatRate { S7_SetPoint := 'True'} : "stCalcValue";   // kW
         DeltaP { S7_SetPoint := 'True'} : "stCalcValue";   // kPa
         TemperatureRateOfChange { S7_SetPoint := 'True'} : "stCalcValue";   // C/s
         Massflow { S7_SetPoint := 'True'} : "stCalcValue";   // Heating media massflow (t/h)
      END_STRUCT;
      HighPressPart : Struct
         CompressorSaturationTemperature : "stCalcValue";
         CompressorSuperheat : "stCalcValue";   // C
         CondenserSaturationTemperature : "stCalcValue";   // C
         CondenserSubcooling : "stCalcValue";   // C
         ExpansionValveSubcooling : "stCalcValue";   // C
         CondenserDeltaP : "stCalcValue";   // kPa
      END_STRUCT;
      LowPressPart : Struct
         EvaporatorSuperheat : "stCalcValue";   // C
         CompressorSuperheat { S7_SetPoint := 'True'} : "stCalcValue";   // C
         EvaporatorSaturationTemperature { S7_SetPoint := 'True'} : "stCalcValue";   // C
         CompressorSaturationTemperature { S7_SetPoint := 'True'} : "stCalcValue";   // C
      END_STRUCT;
      System : Struct
         Quality : "stCalcValue";   // 1
         COP { S7_SetPoint := 'True'} : "stCalcValue";   // 1
         ElectricalPower { S7_SetPoint := 'True'} : "stCalcValue";   // kW
         TemperatureLift { S7_SetPoint := 'True'} : "stCalcValue";   // C
         MotorEfficiency { S7_SetPoint := 'True'} : "stCalcValue";   // Instantaneous efficiency (%)
         FMEP { S7_SetPoint := 'True'} : "stCalcValue";   // kPa
      END_STRUCT;
      Auxiliary : Struct
         ShaftSealDeltaT : "stCalcValue";   // C
         CPCDeltaP { S7_SetPoint := 'True'} : "stCalcValue";
      END_STRUCT;
      Misc : Struct
         EvaporatorDischargePressureMean { S7_SetPoint := 'True'} : "stCalcValue";   // Average of Evaporator A & B discharge pressures
         EvaporatorDischargeTemperatureMin { S7_SetPoint := 'True'} : "stCalcValue";   // Smaller of Evaporator A & B discharge temperatures
         EvaporatorDischargeTemperatureMean { S7_SetPoint := 'True'} : "stCalcValue";   // Average of Evaporator A & B discharge temperatures
         OilFilterDeltaP { S7_SetPoint := 'True'} : "stCalcValue";   // kPa
      END_STRUCT;
   END_VAR
BEGIN
   HeatSink.DeltaP.fMin := 0.0;
   HeatSink.DeltaP.fMax := 1000.0;
   HeatSink.DeltaP.bCheckLimits := TRUE;
   HeatSource.DeltaP.fMax := 4000.0;
   HeatSource.DeltaP.bCheckLimits := true;
END_DATA_BLOCK

DATA_BLOCK "DB_DI"   // DB2
{ S7_Optimized_Access := 'TRUE' }
AUTHOR : Heaten
VERSION : 0.1
// stored: AutoNumber true, DBAccessibleFromOPCUA true, DBAccessibleFromWebserver true, IsOnlyStoredInLoadMemory false, IsRetainMemResEnabled false, IsWriteProtectedInAS false, MemoryReserve 0
   VAR RETAIN
      SafetyRelayStatus { S7_SetPoint := 'True'} : "stDigitalInput";   // Emergency Stop status
      HBL_FS_01 { S7_SetPoint := 'True'} : "stDigitalInput";   // Flow switch heat source
      HBL_FS_02 { S7_SetPoint := 'True'} : "stDigitalInput";   // Flow switch heat sink
      HBL_EC_01_X1 { S7_SetPoint := 'True'} : "stDigitalInput";   // Oil heaters group 1 status
      HBL_EC_02_X1 { S7_SetPoint := 'True'} : "stDigitalInput";   // Oil heaters group 2 status
      DI08 { S7_SetPoint := 'True'} : "stDigitalInput";   // 24V Distribution status
      HBL_PS_500_X2 { S7_SetPoint := 'True'} : "stDigitalInput";   // Compressor discharge manifold A & B high pressure
      HBL_LS_01 { S7_SetPoint := 'True'} : "stDigitalInput";   // Drip pan sump A full
      HBL_LS_02 { S7_SetPoint := 'True'} : "stDigitalInput";   // Drip pan sump B full
      HBL_PZH_539 { S7_SetPoint := 'True'} : "stDigitalInput";   // Evaporator discharge pressure switch
      HBL_LS_632 { S7_SetPoint := 'True'} : "stDigitalInput";   // Oil separator stage 1 oil level high
      HBL_LS_633 { S7_SetPoint := 'True'} : "stDigitalInput";   // Oil separator stage 2 oil level high
      VPNUserConnected { S7_SetPoint := 'True'} : "stDigitalInput";   // VPN user logged in signal from VPN router
      CPC_LS_864 { S7_SetPoint := 'True'} : "stDigitalInput";
      HBL_LS_644 { S7_SetPoint := 'True'} : "stDigitalInput";   // Suction accumulator level switch
      HBL_LS_674 { S7_SetPoint := 'True'} : "stDigitalInput";   // Discharge accumulator level switch
      HBL_HV_640_X1 { S7_SetPoint := 'True'} : "stDigitalInput";   // Suction accumualtor drain valve open status
      HBL_HV_640_X2 { S7_SetPoint := 'True'} : "stDigitalInput";   // Suction accumualtor drain valve closed status
      HBL_HV_670_X1 { S7_SetPoint := 'True'} : "stDigitalInput";   // Discharge accumulator drain valve open status
      HBL_HV_670_X2 { S7_SetPoint := 'True'} : "stDigitalInput";   // Discharge accumulator drain valve closed status
      CPC_HV_852_X1 { S7_SetPoint := 'True'} : "stDigitalInput";   // CPC Cooler enable valve open status
      CPC_HV_852_X2 { S7_SetPoint := 'True'} : "stDigitalInput";   // CPC Cooler enable valve closed status
      HBL_HV_861_X1 { S7_SetPoint := 'True'} : "stDigitalInput";   // Compressor manifold drain valve open status
      HBL_HV_861_X2 { S7_SetPoint := 'True'} : "stDigitalInput";   // Compressor manifold drain valve closed status
   END_VAR
   VAR
      CPC_LSH_870A { S7_SetPoint := 'True'} : "stDigitalInput";   // CPC manifold refrigerant level upper
      CPC_LSL_870B { S7_SetPoint := 'True'} : "stDigitalInput";   // CPC manifold refrigernat level lower
      CPC_PZH_874 { S7_SetPoint := 'True'} : "stDigitalInput";   // CPC manifold pressure switch
   END_VAR
BEGIN
   HBL_PS_500_X2.bValueOnError := true;
END_DATA_BLOCK

DATA_BLOCK "DB_DO"   // DB8
{ S7_Optimized_Access := 'TRUE' }
AUTHOR : Heaten
VERSION : 0.1
// stored: AutoNumber true, DBAccessibleFromOPCUA true, DBAccessibleFromWebserver true, IsOnlyStoredInLoadMemory false, IsRetainMemResEnabled false, IsWriteProtectedInAS false, MemoryReserve 0
   VAR
      DistributionReset : Bool;   // 24V distributon control
      CabinetFan : Bool;   // PLC cabinet fan
      CabinetHeater : Bool;   // PLC cabinet heater
      HBL_EC_01 : Bool;   // Oil pan oil heaters group 1
      HBL_EC_02 : Bool;   // Oil pan oil heaters group 2
      HBL_HV_630 : Bool;   // Oil separator stage 1 oil return valve
      HBL_HV_114 : Bool;   // Suction manifold drain valve L
      HBL_HV_115 : Bool;   // Suction manifold drain valve R
      HBL_HV_860 : Bool;   // CPC tank refrigerant return selection valve
      HBL_HV_861 : Bool;   // Compressor manifold refrigerant return selection valve
      SSC_P_01 : Bool;   // SSC barrier fluid circulation pump
      SSC_F_01 : Bool;   // SSC barrier fluid cooling fan
      SSC_P_02 : Bool;   // SSC barrier fluid recharge pump
      CPC_P_01 : Bool;   // CPC refrigerant reinjection pump
      SpareContactor1 : Bool;
      SpareContactor2 : Bool;
      HBL_HV_631 : Bool;   // Oil separator stage 2 oil return valve
      HBL_HV_640_Y1 : Bool;   // Suction accumualtor drain valve open command
      HBL_HV_640_Y2 : Bool;   // Suction accumualtor drain valve close command
      HBL_HV_670_Y1 : Bool;   // Discharge accumulator drain valve open command
      HBL_HV_670_Y2 : Bool;   // Discharge accumulator drain valve close command
      CPC_HV_852_Y1 : Bool;   // CPC Cooler enable valve open command
      CPC_HV_852_Y2 : Bool;   // CPC Cooler enable valve close command
      HBL_HV_861_Y1 : Bool;   // Compressor manifold drain valve open command
      HBL_HV_861_Y2 : Bool;   // Compressor manifold drain valve close command
      HBL_HV_676 : Bool;   // Discharge accumulator drain valve 2
      HBL_HV_563 : Bool;   // Evaporator 1 axis A valve
      HBL_HV_564 : Bool;   // Evaporator 2 axis A valve
   END_VAR
BEGIN
END_DATA_BLOCK

DATA_BLOCK "DB_InverterDrives"   // DB41
{ S7_Optimized_Access := 'FALSE' }
AUTHOR : Heaten
VERSION : 0.1
// stored: AutoNumber true, DBAccessibleFromOPCUA true, DBAccessibleFromWebserver true, IsOnlyStoredInLoadMemory false, IsWriteProtectedInAS false
   VAR RETAIN
      CPC_SC_01 { S7_SetPoint := 'True'} : "stInverterDrive";   // CPC Cooling fan
      HBL_SC_01 { S7_SetPoint := 'True'} : "stInverterDrive";   // Container ventilation fan
      HBL_SC_02 { S7_SetPoint := 'True'} : "stInverterDrive";   // Compressor lubrication pump
      HBL_SC_03 { S7_SetPoint := 'True'} : "stInverterDrive";   // CPC Pump
      HBL_SC_10 { S7_SetPoint := 'True'} : "stInverterDrive";   // Compressor motor
   END_VAR
BEGIN
   CPC_SC_01.Cmd.Speed.Raw.iMax := 20000;
   CPC_SC_01.Cmd.Speed.Eng.fMax := 1500.0;
   CPC_SC_01.Cmd.Torque.Raw.iMax := 10000;
   CPC_SC_01.Cmd.Torque.Eng.fMax := 100.0;
   CPC_SC_01.Stat.Speed.Raw.iMax := 20000;
   CPC_SC_01.Stat.Speed.Eng.fMax := 1500.0;
   CPC_SC_01.Stat.Torque.Raw.iMax := 10000;
   CPC_SC_01.Stat.Torque.Eng.fMax := 100.0;
   CPC_SC_01.Stat.Power.Raw.iMax := 10000;
   CPC_SC_01.Stat.Power.Eng.fMax := 1.5;
   HBL_SC_01.Cmd.Speed.Raw.iMax := 20000;
   HBL_SC_01.Cmd.Speed.Eng.fMin := 0.0;
   HBL_SC_01.Cmd.Speed.Eng.fMax := 1500.0;
   HBL_SC_01.Cmd.Torque.Raw.iMax := 10000;
   HBL_SC_01.Cmd.Torque.Eng.fMax := 100.0;
   HBL_SC_01.Stat.Speed.Raw.iMax := 20000;
   HBL_SC_01.Stat.Speed.Eng.fMax := 1500.0;
   HBL_SC_01.Stat.Torque.Raw.iMax := 10000;
   HBL_SC_01.Stat.Torque.Eng.fMax := 100.0;
   HBL_SC_01.Stat.Power.Raw.iMax := 10000;
   HBL_SC_01.Stat.Power.Eng.fMax := 1.5;
   HBL_SC_02.Cmd.Speed.Raw.iMax := 20000;
   HBL_SC_02.Cmd.Speed.Eng.fMax := 5000.0;
   HBL_SC_02.Cmd.Torque.Raw.iMax := 10000;
   HBL_SC_02.Cmd.Torque.Eng.fMax := 100.0;
   HBL_SC_02.Stat.Speed.Raw.iMax := 20000;
   HBL_SC_02.Stat.Speed.Eng.fMax := 5000.0;
   HBL_SC_02.Stat.Torque.Raw.iMax := 10000;
   HBL_SC_02.Stat.Torque.Eng.fMax := 100.0;
   HBL_SC_02.Stat.Power.Raw.iMax := 10000;
   HBL_SC_02.Stat.Power.Eng.fMax := 2.0;
   HBL_SC_03.Cmd.Speed.Raw.iMax := 20000;
   HBL_SC_03.Cmd.Speed.Eng.fMax := 1500.0;
   HBL_SC_03.Cmd.Torque.Raw.iMax := 10000;
   HBL_SC_03.Cmd.Torque.Eng.fMax := 100.0;
   HBL_SC_03.Stat.Speed.Raw.iMax := 20000;
   HBL_SC_03.Stat.Speed.Eng.fMax := 1500.0;
   HBL_SC_03.Stat.Torque.Raw.iMax := 10000;
   HBL_SC_03.Stat.Torque.Eng.fMax := 100.0;
   HBL_SC_03.Stat.Power.Raw.iMax := 10000;
   HBL_SC_03.Stat.Power.Eng.fMax := 2.0;
   HBL_SC_10.Cmd.Speed.Raw.iMin := 0;
   HBL_SC_10.Cmd.Speed.Raw.iMax := 20000;
   HBL_SC_10.Cmd.Speed.Eng.fMin := 0.0;
   HBL_SC_10.Cmd.Speed.Eng.fMax := 1500.0;
   HBL_SC_10.Cmd.Torque.Raw.iMin := 0;
   HBL_SC_10.Cmd.Torque.Raw.iMax := 10000;
   HBL_SC_10.Cmd.Torque.Eng.fMin := 0.0;
   HBL_SC_10.Cmd.Torque.Eng.fMax := 100.0;
   HBL_SC_10.Stat.Speed.Raw.iMax := 20000;
   HBL_SC_10.Stat.Speed.Eng.fMin := 0.0;
   HBL_SC_10.Stat.Speed.Eng.fMax := 1500.0;
   HBL_SC_10.Stat.Torque.Raw.iMin := 0;
   HBL_SC_10.Stat.Torque.Raw.iMax := 10000;
   HBL_SC_10.Stat.Torque.Eng.fMin := 0.0;
   HBL_SC_10.Stat.Torque.Eng.fMax := 100.0;
   HBL_SC_10.Stat.Power.Raw.iMin := 0;
   HBL_SC_10.Stat.Power.Raw.iMax := 10000;
   HBL_SC_10.Stat.Power.Eng.fMin := 0.0;
   HBL_SC_10.Stat.Power.Eng.fMax := 1000.0;
END_DATA_BLOCK

DATA_BLOCK "DB_Misc"   // DB6
{ S7_Optimized_Access := 'TRUE' }
AUTHOR : Heaten
VERSION : 0.1
// stored: AutoNumber true, DBAccessibleFromOPCUA true, DBAccessibleFromWebserver true, IsOnlyStoredInLoadMemory false, IsRetainMemResEnabled false, IsWriteProtectedInAS false, MemoryReserve 100
   VAR
      EvaporatorDischargePressureMean : "stCalcSelect";   // Average of Evaporator A & B discharge pressures
      EvaporatorDischargeTemperatureMin { S7_SetPoint := 'True'} : "stCalcSelect";   // Smaller of Evaporator A & B discharge temperatures
      EvaporatorDischargeTemperatureMean { S7_SetPoint := 'True'} : "stCalcSelect";   // Average of Evaporator A & B discharge temperatures
      EvaporatorDischargePressureOffset : Real := 0.0;   // HBL-PT-04
   END_VAR
BEGIN
   EvaporatorDischargePressureMean.nMode := 5;
   EvaporatorDischargeTemperatureMin.nMode := 3;
   EvaporatorDischargeTemperatureMean.nMode := 5;
END_DATA_BLOCK

DATA_BLOCK "DB_Profiling"   // DB100
{ S7_Optimized_Access := 'TRUE' }
AUTHOR : Heaten
VERSION : 0.1
// stored: AutoNumber false, DBAccessibleFromOPCUA true, DBAccessibleFromWebserver true, IsOnlyStoredInLoadMemory false, IsRetainMemResEnabled false, IsWriteProtectedInAS false, MemoryReserve 100
   VAR
      OB1time : "stProfile";
      OB30time { S7_SetPoint := 'True'} : "stProfile";
      Section10time : "stProfile";
      Section20time : "stProfile";
      Section30time : "stProfile";
      Section40time : "stProfile";
      Section60time : "stProfile";
      Section80time : "stProfile";
      Section90time : "stProfile";
      Section10_DigitalInputProcessing { S7_SetPoint := 'True'} : "stProfile";
      Section10_AnalogInputProcessing { S7_SetPoint := 'True'} : "stProfile";
      Section10_InverterDriveProcessing { S7_SetPoint := 'True'} : "stProfile";
      Section10_InputAlarmHandling { S7_SetPoint := 'True'} : "stProfile";
      Section20_Calculations { S7_SetPoint := 'True'} : "stProfile";
      Section20_StateMachine { S7_SetPoint := 'True'} : "stProfile";
      Section20_ControlAlarmHandling { S7_SetPoint := 'True'} : "stProfile";
      Section20_Regulation { S7_SetPoint := 'True'} : "stProfile";
      Section20_StartStopControl { S7_SetPoint := 'True'} : "stProfile";
   END_VAR
BEGIN
END_DATA_BLOCK

DATA_BLOCK "DB_Regulators"   // DB18
{ S7_Optimized_Access := 'FALSE' }
AUTHOR : Heaten
VERSION : 0.1
// stored: AutoNumber true, DBAccessibleFromOPCUA true, DBAccessibleFromWebserver true, IsOnlyStoredInLoadMemory false, IsWriteProtectedInAS false
   VAR RETAIN
      CabinetTemperature : "stTemperatureController2";   // Regulates PLC cabinet temperature
      OilHeating { S7_SetPoint := 'True'} : "stOilHeater";   // Regulates compressor oil sump temperature
      ContainerVentilation { S7_SetPoint := 'True'} : "stPI_Regulator";   // Regulates container air temperature
      CPCPressure { S7_SetPoint := 'True'} : "stPI_Regulator";   // Regulates CPC pressure
      CPCReservoir { S7_SetPoint := 'True'} : "stOnOffRegulator";   // Regulates CPC reservoir level
      CPCReservoirPlanB { S7_SetPoint := 'True'} : "stProgressivePeriodicRegulator4";   // Regulates CPC reservoir level (Plan B)
      ShaftSealCirculation { S7_SetPoint := 'True'} : "stCirculationPump";   // Barrier fluid circulation
      ShaftSealCooler { S7_SetPoint := 'True'} : "stOnOffRegulator";   // Barrier fluid temperature
      ShaftSealRecharge { S7_SetPoint := 'True'} : "stOnOffRegulator";   // Barrier fluid pressure
      OilSeparator { S7_SetPoint := 'True'} : "stOilSeparator";   // Regulates oil level in oil separator
      LubricationPriming { S7_SetPoint := 'True'} : "stPrimerPump";   // Compressor lubrication priming
      PerformanceControl { S7_SetPoint := 'True'} : "stPerformanceControl";   // Compressor speed control
      SuperheatControl { S7_SetPoint := 'True'} : "stSuperheatControl";   // Regulates superheat
      PinchControl { S7_SetPoint := 'True'} : "stPinchControl";   // Regulates pinch
      PurgeControl { S7_SetPoint := 'True'} : "stPurgeControl";   // Handles purging of compressor suction manifold
      FilterDryer { S7_SetPoint := 'True'} : "stFilterDryer";   // Runs filter dryer circuit
      OilRecovery { S7_SetPoint := 'True'} : "stOilRecovery";   // Runs oil recovery circuit
      RecuperatorBypass { S7_SetPoint := 'True'} : "stNullRegulator";   // Runs recuperator bypass
      HeatSourceCycle { S7_SetPoint := 'True'} : "stTrackingRegulator";
      HeatSourceCyclePIP { S7_SetPoint := 'True'} : "stPIP_Regulator";   // Regulates heat exchanger temperature rise
      DischargeAccumulator { S7_SetPoint := 'True'} : "stOnOffRegulator3";   // Discharge accumulator return
      SuctionAccumulator { S7_SetPoint := 'True'} : "stOnOffRegulator3";   // Suction accumulator return
      HeatboosterSetpoint { S7_SetPoint := 'True'} : Real;   // TEST: selected setpoint
      RegulationTarget : Int;   // TEST: selected regulation target
   END_VAR
BEGIN
   CabinetTemperature.bEnable := true;
   CabinetTemperature.fHeatingSetpoint := 15.0;
   CabinetTemperature.fCoolingSetpoint := 40.0;
   OilHeating.fOilSuperheat := 15.0;
   OilHeating.Controller.bEnable := true;
   OilHeating.Controller.fHysteresis := 2.0;
   ContainerVentilation.bEnable := false;
   CPCPressure.bEnable := false;
   CPCReservoir.bEnable := true;
   CPCReservoir.fSetpoint := 60.0;
   CPCReservoirPlanB.tManualPeriod := T#10m;
   CPCReservoirPlanB.tOnTime := T#15s;
   CPCReservoirPlanB.Param.Limit[0] := 400.0;
   CPCReservoirPlanB.Param.Limit[1] := 500.0;
   CPCReservoirPlanB.Param.Limit[2] := 600.0;
   CPCReservoirPlanB.Param.Limit[3] := 700.0;
   CPCReservoirPlanB.Param.Period[0] := T#20m;
   CPCReservoirPlanB.Param.Period[1] := T#14m;
   CPCReservoirPlanB.Param.Period[2] := T#7m;
   CPCReservoirPlanB.Param.Period[3] := T#1m;
   ShaftSealCirculation.bEnable := true;
   ShaftSealCooler.bEnable := true;
   ShaftSealCooler.fSetpoint := 97.5;
   ShaftSealCooler.fHysteresis := 5.0;
   ShaftSealRecharge.bEnable := true;
   ShaftSealRecharge.fSetpoint := 1120.0;
   ShaftSealRecharge.fHysteresis := 200.0;
   // OilSeparator.Stage1 : Level control Stage 1
   // OilSeparator.Stage2 : Level control Stage 2
   LubricationPriming.fMotorSpeed := 2830.0;
   LubricationPriming.fMotorTorqueLimit := 70.0;
   LubricationPriming.Controller.bEnable := true;
   LubricationPriming.Controller.fSetpoint := 140.0;
   LubricationPriming.Controller.fHysteresis := 80.0;
   PerformanceControl.Settings.HeatSink.Control_Active := true;
   PerformanceControl.Settings.HeatSink.Kp := 16.0;
   PerformanceControl.Settings.HeatSource.Control_Active := false;
   PerformanceControl.Settings.HeatSource.Kp := -4.0;
   PerformanceControl.Settings.VariableControl.Control_Active := false;
   PerformanceControl.Settings.Config.MinimumPerformanceRequirement := 30.0;
   PerformanceControl.Settings.Config.MaximumAdditionalSuperheat := 35.0;
   PerformanceControl.Settings.Config.INCREASEWITHNORESTRICTION := 0.2;
   SuperheatControl.bEnable := true;
   SuperheatControl.Regulator.fFeedbackHysteresis := 15.0;
   SuperheatControl.Regulator.fOutMax := 100.0;
   SuperheatControl.Regulator.fOutMin := -50.0;
   SuperheatControl.Regulator.Kp := 0.8;
   SuperheatControl.Regulator.Tn := 35.0;
   SuperheatControl.Regulator.Tv := 0.0;
   SuperheatControl.Regulator.T1 := 0.0;
   SuperheatControl.fineTuningRecTarget := 0.65;
   SuperheatControl.ExponentialPinchFactor := 21.6;
   PinchControl.bEnable := true;
   PinchControl.Regulator.fOutMax := 100.0;
   PinchControl.Regulator.Kp := 1.0;
   PinchControl.Regulator.Tn := 4.0;
   PinchControl.Regulator.Tv := 16.0;
   PinchControl.Regulator.T1 := 0.0;
   PurgeControl.nPurgeCycles := 3;
   PurgeControl.bEnable := true;
   PurgeControl.Purge.nPurgeType := 0;
   PurgeControl.Purge.tPurgeTime := T#15s;
   PurgeControl.Purge.fPurgeDeltaP := 35.0;
   PurgeControl.Spin.tSpinTime := T#20s;
   PurgeControl.Spin.fSpinSpeed := 250.0;
   PurgeControl.Spin.fSpinRamp := 50.0;
   FilterDryer.fFixedOutput := 50.0;
   FilterDryer.Controller.tOnTime := T#3m;
   FilterDryer.Controller.tPeriod := T#30m;
   OilRecovery.nRunRatio := 5;
   OilRecovery.Controller.tOnTime := T#1m;
   OilRecovery.Controller.tStartDelay := T#5s;
   // HeatSourceCyclePIP.fPV : [C] Heat source temperature
   // HeatSourceCyclePIP.fPVvel : [K/sec] Heat source temperature rate of change
   HeatSourceCyclePIP.fSP := 120.0;   // [C] Heat source temperature setpoint
   HeatSourceCyclePIP.fOutMax := 100.0;   // [%] Max valve position
   HeatSourceCyclePIP.fOutMin := 0.0;   // [%] Min valve position
   HeatSourceCyclePIP.fVelMax := 5.0;   // [K/min] Max positive temperature rate of change
   HeatSourceCyclePIP.fVelMin := -5.0;   // [K/min] Max negative temperature rate of change
   // HeatSourceCyclePIP.fOut : [%] Valve position
   // HeatSourceCyclePIP.fManualValue : [%] Manual manipulated value
   HeatSourceCyclePIP.Kp := 1.0;   // Proportional gain temperature (C/s per C)
   HeatSourceCyclePIP.Tn := 0.0;   // Integral gain temperature
   HeatSourceCyclePIP.KpVel := 15.0;   // Proportional gain temperature rate of change (% per C/s)
   HeatSourceCyclePIP.TnVel := 75.0;
   HeatSourceCyclePIP.fFeedbackHysteresis := 0.2;
END_DATA_BLOCK

DATA_BLOCK "DB_State"   // DB12
{ S7_Optimized_Access := 'TRUE' }
AUTHOR : Heaten
VERSION : 0.1
// stored: AutoNumber true, DBAccessibleFromOPCUA true, DBAccessibleFromWebserver true, IsOnlyStoredInLoadMemory false, IsRetainMemResEnabled false, IsWriteProtectedInAS false, MemoryReserve 100
   VAR
      SystemInitialised : Bool;
      StopRequired : Bool;
      FastStop : Bool;
      StopLock : Bool;   // Not used
      ForceStateChangeFlags : Array[1..16] of Bool;
      RunningConditions : Struct
         ShaftSealSystemOK : Bool;
         OilHeatOK : Bool;
         HeatSinkTemperatureOK : Bool;
         HeatSourceTemperatureOK : Bool;
         SuperheatCompressorInOK : Bool;
         PressureSpreadOK : Bool;
         SuperheatCompressorOutOK : Bool;
         RecuperatorWorking : Bool;
         AtOrAboveHydrolockSpeed : Bool;
         SuctionLineDry : Bool;
         AuxiliariesOK : Bool;
         HeatSourceFlowOK : Bool;
         HeatSinkFlowOK : Bool;
         LubricationPrimingOk : Bool;
         DoWarmStart : Bool;
         CompressorStopped : Bool;
         RiskOfHydrolock : Bool;
      END_STRUCT;
      State : Struct
         State_Number : Int := -1;
         "0_Initialisation" : Bool;
         "1_Offline" : Bool;
         "2_Standby" : Bool;
         "3_PrepareStart" : Bool;
         "4_Start" : Bool;
         "5_Warmup" : Bool;
         "6_Running" : Bool;
         "7_Stop" : Bool;
      END_STRUCT;
      StatePauseFlags { S7_SetPoint := 'True'} : Array[0..7] of Bool;   // Allow pausing (level signal)
      StateConfirmFlags : Array[0..7] of Bool;   // Confirm past pause (momentary signal)
      StateDwellTimeElapsed : Array[0..8] of Bool;
   END_VAR
BEGIN
END_DATA_BLOCK

DATA_BLOCK "DB_System"   // DB42
{ S7_Optimized_Access := 'TRUE' }
AUTHOR : Heaten
VERSION : 0.1
// stored: AutoNumber true, DBAccessibleFromOPCUA true, DBAccessibleFromWebserver true, IsOnlyStoredInLoadMemory false, IsRetainMemResEnabled false, IsWriteProtectedInAS false, MemoryReserve 100
   VAR
      bFirstCycle : Bool := FALSE;   // High on first scan only
      bFirstCycleCyclic : Bool := FALSE;
      bSimulation : Bool := FALSE;   // Simulation active
      bProfiling : Bool := FALSE;   // Profiling active
      bInternalEmergencyStop : Bool := FALSE;   // PLC source E-stop. 0 = ok, 1 = Emergency stop
      bExternalEmergencyStop : Bool := FALSE;   // External source E-stop. 0 = ok, 1 = Emergency stop
      bEmergencyStop : Bool := FALSE;   // Emergency stop state. 0 = ok, 1 = Emergency stop
      bManualModeWarning : Bool := FALSE;   // 1 = one or more regulators in manual mode, 0 = no regulators in manual mode
      bExternalValidData { S7_SetPoint := 'True'} : Bool := TRUE;   // 1 = values sent from APP PLC are valid
      fCycleTime : Real := 0.1000159;   // Cycle time in sec
      lfCycleTime : LReal := 0.100015944;   // Cycle time in sec
      BarometricOffset : Real := 101.325;   // [kPa] Pressure offset relative to absolute
   END_VAR
   VAR RETAIN
      SystemUptime : "stHoursCounter";   // System powered on
      SystemActiveTime { S7_SetPoint := 'True'} : "stHoursCounter";   // Standby or higher
      RunningTime { S7_SetPoint := 'True'} : "stHoursCounter";   // In running state
   END_VAR
   VAR
      SafetyRelay { S7_SetPoint := 'True'} : "stSafetyRelay";   // Emergency stop safety relay
      WinCCLink { S7_SetPoint := 'True'} : "stHeartbeat";
   END_VAR
   VAR RETAIN
      AppPLCLink { S7_SetPoint := 'True'} : "stHeartbeatCount2";
   END_VAR
   VAR
      SoftwareVersion : String := 'V4.0.0.6';   // PLC software version string (set in FC35)
   END_VAR
BEGIN
   SystemUptime.nHours := 5956;
   SystemUptime.nMinutes := 7;
   SystemUptime.nSeconds := 43;
   SystemUptime.bReset := FALSE;
   SystemActiveTime.nHours := 0;
   SystemActiveTime.nMinutes := 0;
   SystemActiveTime.nSeconds := 0;
   SystemActiveTime.bReset := FALSE;
   RunningTime.nHours := 0;
   RunningTime.nMinutes := 0;
   RunningTime.nSeconds := 0;
   RunningTime.bReset := FALSE;
   SafetyRelay.tResetLoopTime := T#1S;
   SafetyRelay.tResetTimeout := T#1S;
   SafetyRelay.nState := 3;
   SafetyRelay.bStatus := TRUE;
   SafetyRelay.bResetReq := FALSE;
   SafetyRelay.bResetLoop := FALSE;
   SafetyRelay.bResetCmd := FALSE;
   SafetyRelay.bResetFailed := FALSE;
   WinCCLink.bOut := FALSE;
   WinCCLink.bIn := TRUE;
   WinCCLink.bEnable := TRUE;
   WinCCLink.bOk := TRUE;
   WinCCLink.nState := 2;
   WinCCLink.tTimeout := T#1M_30S;
   AppPLCLink.nLocalCount := 0;
   AppPLCLink.nRemoteCount := 35505;
   AppPLCLink.bEnable := TRUE;
   AppPLCLink.bOk := TRUE;
   AppPLCLink.nState := 2;
   AppPLCLink.tTimeout := T#2S;
END_DATA_BLOCK

DATA_BLOCK "DB_Valves"   // DB46
{ S7_Optimized_Access := 'FALSE' }
AUTHOR : Heaten
VERSION : 0.1
// stored: AutoNumber false, DBAccessibleFromOPCUA true, DBAccessibleFromWebserver true, IsOnlyStoredInLoadMemory false, IsWriteProtectedInAS false
   VAR RETAIN
      HBL_HCV_576 : "stRegulatingValve";   // Expansion Valve A
      HBL_HCV_578 : "stRegulatingValve";   // Expansion Valve B
      HBL_HCV_577 { S7_SetPoint := 'True'} : "stRegulatingValve";   // Expansion Valve A2
      HBL_HCV_579 { S7_SetPoint := 'True'} : "stRegulatingValve";   // Expansion Valve B2
      HBL_HCV_515 { S7_SetPoint := 'True'} : "stRegulatingValve";   // Heat sink condensate blowdown flow control valve
      HBL_HCV_575 { S7_SetPoint := 'True'} : "stRegulatingValve";   // Recuperator oil drain valve
      HBL_HCV_616 { S7_SetPoint := 'True'} : "stRegulatingValve";   // Recuperator bypass valve
      HBL_HCV_700 { S7_SetPoint := 'True'} : "stRegulatingValve";   // Oil recovery refrigerant blowdown valve
      HBL_HCV_514 { S7_SetPoint := 'True'} : "stRegulatingValve";   // Heat sink discharge pressure control valve
      HBL_HCV_548 { S7_SetPoint := 'True'} : "stRegulatingValve";   // Heat source suction pressure control valve
      CPC_HCV_853 { S7_SetPoint := 'True'} : "stRegulatingValve";   // CPC cooler water control valve
      CPC_HCV_880 { S7_SetPoint := 'True'} : "stRegulatingValve";   // CPC subcooler water control valve
      HBL_HCV_900 { S7_SetPoint := 'True'} : "stRegulatingValve";   // Heat sink condensate feed valve
      HBL_HV_640 { S7_SetPoint := 'True'} : "stProcessValve2";   // Suction accumulator drain valve
      HBL_HV_670 { S7_SetPoint := 'True'} : "stProcessValve2";   // Discharge accumulator drain valve
      CPC_HV_852 { S7_SetPoint := 'True'} : "stProcessValve2";   // CPC cooler enable valve
      HBL_HV_861 { S7_SetPoint := 'True'} : "stProcessValve2";   // Compressor manifold drain valve
   END_VAR
BEGIN
   // HBL_HCV_576.Cmd.Position : Expansion Valve A
   HBL_HCV_576.Cmd.Position.Raw.iMax := 27648;
   HBL_HCV_576.Cmd.Position.Eng.fMin := 0.0;
   HBL_HCV_576.Cmd.Position.Eng.fMax := 100.0;
   // HBL_HCV_576.Stat.Position : Expansion Valve A
   HBL_HCV_576.Stat.Position.Raw.iMin := 0;
   HBL_HCV_576.Stat.Position.Raw.iMax := 27648;
   HBL_HCV_576.Stat.Position.Eng.fMin := 0.0;
   HBL_HCV_576.Stat.Position.Eng.fMax := 100.0;
   // HBL_HCV_578.Cmd.Position : Expansion Valve B
   HBL_HCV_578.Cmd.Position.Raw.iMin := 0;
   HBL_HCV_578.Cmd.Position.Raw.iMax := 27648;
   HBL_HCV_578.Cmd.Position.Eng.fMin := 0.0;
   HBL_HCV_578.Cmd.Position.Eng.fMax := 100.0;
   // HBL_HCV_578.Stat.Position : Expansion Valve B
   HBL_HCV_578.Stat.Position.Raw.iMin := 0;
   HBL_HCV_578.Stat.Position.Raw.iMax := 27648;
   HBL_HCV_578.Stat.Position.Eng.fMin := 0.0;
   HBL_HCV_578.Stat.Position.Eng.fMax := 100.0;
   HBL_HCV_577.Cmd.Position.Raw.iMin := 0;
   HBL_HCV_577.Cmd.Position.Raw.iMax := 27648;
   HBL_HCV_577.Cmd.Position.Eng.fMin := 0.0;
   HBL_HCV_577.Cmd.Position.Eng.fMax := 100.0;
   HBL_HCV_577.Stat.Position.Raw.iMin := 0;
   HBL_HCV_577.Stat.Position.Raw.iMax := 27648;
   HBL_HCV_577.Stat.Position.Eng.fMin := 0.0;
   HBL_HCV_577.Stat.Position.Eng.fMax := 100.0;
   HBL_HCV_579.Cmd.Position.Raw.iMin := 0;
   HBL_HCV_579.Cmd.Position.Raw.iMax := 27648;
   HBL_HCV_579.Cmd.Position.Eng.fMin := 0.0;
   HBL_HCV_579.Cmd.Position.Eng.fMax := 100.0;
   HBL_HCV_579.Stat.Position.Raw.iMin := 0;
   HBL_HCV_579.Stat.Position.Raw.iMax := 27648;
   HBL_HCV_579.Stat.Position.Eng.fMin := 0.0;
   HBL_HCV_579.Stat.Position.Eng.fMax := 100.0;
   HBL_HCV_515.Cmd.Position.Raw.iMin := 0;
   HBL_HCV_515.Cmd.Position.Raw.iMax := 27648;
   HBL_HCV_515.Cmd.Position.Eng.fMin := 0.0;
   HBL_HCV_515.Cmd.Position.Eng.fMax := 100.0;
   HBL_HCV_515.Stat.Position.Raw.iMin := 0;
   HBL_HCV_515.Stat.Position.Raw.iMax := 27648;
   HBL_HCV_515.Stat.Position.Eng.fMin := 0.0;
   HBL_HCV_515.Stat.Position.Eng.fMax := 100.0;
   HBL_HCV_575.Cmd.Position.Raw.iMin := 0;
   HBL_HCV_575.Cmd.Position.Raw.iMax := 27648;
   HBL_HCV_575.Cmd.Position.Eng.fMin := 0.0;
   HBL_HCV_575.Cmd.Position.Eng.fMax := 100.0;
   HBL_HCV_575.Stat.Position.Raw.iMin := 0;
   HBL_HCV_575.Stat.Position.Raw.iMax := 27648;
   HBL_HCV_575.Stat.Position.Eng.fMin := 0.0;
   HBL_HCV_575.Stat.Position.Eng.fMax := 100.0;
   HBL_HCV_616.Cmd.Position.Raw.iMin := 0;
   HBL_HCV_616.Cmd.Position.Raw.iMax := 27648;
   HBL_HCV_616.Cmd.Position.Eng.fMin := 0.0;
   HBL_HCV_616.Cmd.Position.Eng.fMax := 100.0;
   HBL_HCV_616.Stat.Position.Raw.iMin := 0;
   HBL_HCV_616.Stat.Position.Raw.iMax := 27648;
   HBL_HCV_616.Stat.Position.Eng.fMin := 0.0;
   HBL_HCV_616.Stat.Position.Eng.fMax := 0.0;
   HBL_HCV_700.Cmd.Position.Raw.iMin := 0;
   HBL_HCV_700.Cmd.Position.Raw.iMax := 27648;
   HBL_HCV_700.Cmd.Position.Eng.fMin := 0.0;
   HBL_HCV_700.Cmd.Position.Eng.fMax := 100.0;
   HBL_HCV_700.Stat.Position.Raw.iMin := 0;
   HBL_HCV_700.Stat.Position.Raw.iMax := 27648;
   HBL_HCV_700.Stat.Position.Eng.fMin := 0.0;
   HBL_HCV_700.Stat.Position.Eng.fMax := 100.0;
   HBL_HCV_548.Cmd.Position.Raw.iMin := 0;
   HBL_HCV_548.Cmd.Position.Raw.iMax := 27648;
   HBL_HCV_548.Cmd.Position.Eng.fMin := 0.0;
   HBL_HCV_548.Cmd.Position.Eng.fMax := 100.0;
   HBL_HCV_548.Stat.Position.Raw.iMin := 0;
   HBL_HCV_548.Stat.Position.Raw.iMax := 27648;
   HBL_HCV_548.Stat.Position.Eng.fMin := 0.0;
   HBL_HCV_548.Stat.Position.Eng.fMax := 100.0;
   CPC_HCV_853.Cmd.Position.Eng.fMax := 100.0;
   CPC_HCV_853.Stat.Position.Eng.fMax := 100.0;
   CPC_HCV_880.Cmd.Position.Eng.fMax := 100.0;
   CPC_HCV_880.Stat.Position.Eng.fMax := 100.0;
END_DATA_BLOCK

DATA_BLOCK "DB_WinCCAlarms"   // DB29
{ S7_Optimized_Access := 'TRUE' }
AUTHOR : Heaten
VERSION : 0.1
// stored: AutoNumber true, DBAccessibleFromOPCUA true, DBAccessibleFromWebserver true, IsOnlyStoredInLoadMemory false, IsRetainMemResEnabled false, IsWriteProtectedInAS false, MemoryReserve 0
   VAR
      "0-System" : Struct
         "0001_WatchdogTimeoutOB1" { S7_SetPoint := 'True'} : "stWinCCAlarm";
         "0003_InitCurrenSettingsFailed" { S7_SetPoint := 'True'} : "stWinCCAlarm";
         "0006_CPUinErrorState" { S7_SetPoint := 'True'} : "stWinCCAlarm";
      END_STRUCT;
      "1-IO" : Struct
         "1001_ConnectionToWinCClost" { S7_SetPoint := 'True'} : "stWinCCAlarm";
         "1002_EmergencyStopActive" { S7_SetPoint := 'True'} : "stWinCCAlarm";
         "1003_SafetyRelayResetFailed" { S7_SetPoint := 'True'} : "stWinCCAlarm";
         "1004_HBL_PS_01_X2" { S7_SetPoint := 'True'} : "stWinCCAlarm";
         "1101_HBL_SC_01_CommError" { S7_SetPoint := 'True'} : "stWinCCAlarm";
         "1102_HBL_SC_02_CommError" { S7_SetPoint := 'True'} : "stWinCCAlarm";
         "1103_HBL_SC_03_CommError" { S7_SetPoint := 'True'} : "stWinCCAlarm";
         "1110_HBL_SC_10_CommError" { S7_SetPoint := 'True'} : "stWinCCAlarm";
         "1121_HBL_SC_01_Tripped" { S7_SetPoint := 'True'} : "stWinCCAlarm";
         "1122_HBL_SC_02_Tripped" { S7_SetPoint := 'True'} : "stWinCCAlarm";
         "1123_HBL_SC_03_Tripped" { S7_SetPoint := 'True'} : "stWinCCAlarm";
         "1130_HBL_SC_10_Tripped" { S7_SetPoint := 'True'} : "stWinCCAlarm";
         "1140_HBL_SC_01_RunFailure" { S7_SetPoint := 'True'} : "stWinCCAlarm";
         "1142_HBL_SC_02_RunFailure" { S7_SetPoint := 'True'} : "stWinCCAlarm";
         "1143_HBL_SC_03_RunFailure" { S7_SetPoint := 'True'} : "stWinCCAlarm";
         "1150_HBL_SC_10_RunFailure" { S7_SetPoint := 'True'} : "stWinCCAlarm";
         "1201_HBL_PT_01_Fault" { S7_SetPoint := 'True'} : "stWinCCAlarm";
         "1202_HBL_PT_02_Fault" { S7_SetPoint := 'True'} : "stWinCCAlarm";
         "1203_HBL_PT_03_Fault" { S7_SetPoint := 'True'} : "stWinCCAlarm";
         "1204_HBL_PT_04_Fault" { S7_SetPoint := 'True'} : "stWinCCAlarm";
         "1205_HBL_TT_05_Fault" { S7_SetPoint := 'True'} : "stWinCCAlarm";
         "1206_HBL_TT_06_Fault" { S7_SetPoint := 'True'} : "stWinCCAlarm";
         "1207_HBL_TT_07_Fault" { S7_SetPoint := 'True'} : "stWinCCAlarm";
         "1208_HBL_TT_08_Fault" { S7_SetPoint := 'True'} : "stWinCCAlarm";
         "1209_HBL_HCV_01_A1_Fault" { S7_SetPoint := 'True'} : "stWinCCAlarm";
         "1210_HBL_TT_10_Fault" { S7_SetPoint := 'True'} : "stWinCCAlarm";
         "1212_HBL_TT_12_Fault" { S7_SetPoint := 'True'} : "stWinCCAlarm";
         "1213_HBL_TT_13_Fault" { S7_SetPoint := 'True'} : "stWinCCAlarm";
         "1214_HBL_TT_14_Fault" { S7_SetPoint := 'True'} : "stWinCCAlarm";
         "1215_HBL_TT_15_Fault" { S7_SetPoint := 'True'} : "stWinCCAlarm";
         "1216_HBL_TT_16_Fault" { S7_SetPoint := 'True'} : "stWinCCAlarm";
         "1217_HBL_TT_17_Fault" { S7_SetPoint := 'True'} : "stWinCCAlarm";
         "1218_HBL_TT_18_Fault" { S7_SetPoint := 'True'} : "stWinCCAlarm";
         "1220_HBL_PT_960_Fault" { S7_SetPoint := 'True'} : "stWinCCAlarm";
         "1221_HBL_PT_05_Fault" { S7_SetPoint := 'True'} : "stWinCCAlarm";
         "1223_HBL_TT_03_Fault" { S7_SetPoint := 'True'} : "stWinCCAlarm";
         "1224_HBL_TT_23_Fault" { S7_SetPoint := 'True'} : "stWinCCAlarm";
         "1225_HBL_TT_24_Fault" { S7_SetPoint := 'True'} : "stWinCCAlarm";
         "1226_HBL_TT_25_Fault" { S7_SetPoint := 'True'} : "stWinCCAlarm";
         "1227_HBL_LT_01_Fault" { S7_SetPoint := 'True'} : "stWinCCAlarm";
         "1228_HBL_TT_21_Fault" { S7_SetPoint := 'True'} : "stWinCCAlarm";
         "1229_HBL_TT_22_Fault" { S7_SetPoint := 'True'} : "stWinCCAlarm";
         "1230_HBL_LT_02_Fault" { S7_SetPoint := 'True'} : "stWinCCAlarm";
         "1231_HBL_HCV_02_A1_Fault" { S7_SetPoint := 'True'} : "stWinCCAlarm";
         "1232_HBL_PT_13_Fault" { S7_SetPoint := 'True'} : "stWinCCAlarm";
         "1233_HBL_TT_20_Fault" { S7_SetPoint := 'True'} : "stWinCCAlarm";
         "1234_HBL_PT_14_Fault" { S7_SetPoint := 'True'} : "stWinCCAlarm";
         "1235_HBL_PT_18_Fault" { S7_SetPoint := 'True'} : "stWinCCAlarm";
         "1236_HBL_PT_19_Fault" { S7_SetPoint := 'True'} : "stWinCCAlarm";
         "1237_HBL_PT_25_Fault" { S7_SetPoint := 'True'} : "stWinCCAlarm";
         "1238_HBL_TT_31_Fault" { S7_SetPoint := 'True'} : "stWinCCAlarm";
         "1239_HBL_TT_33_Fault" { S7_SetPoint := 'True'} : "stWinCCAlarm";
         "1240_HBL_TT_35_Fault" { S7_SetPoint := 'True'} : "stWinCCAlarm";
         "1241_HBL_HCV_01_Fault" { S7_SetPoint := 'True'} : "stWinCCAlarm";
         "1242_HBL_HCV_02_Fault" { S7_SetPoint := 'True'} : "stWinCCAlarm";
         "1243_HBL_PT_07_Fault" { S7_SetPoint := 'True'} : "stWinCCAlarm";
         "1244_HBL_PT_08_Fault" { S7_SetPoint := 'True'} : "stWinCCAlarm";
         "1245_HBL_PT_09_Fault" { S7_SetPoint := 'True'} : "stWinCCAlarm";
         "1246_HBL_PT_10_Fault" { S7_SetPoint := 'True'} : "stWinCCAlarm";
         "1247_HBL_PT_11_Fault" { S7_SetPoint := 'True'} : "stWinCCAlarm";
         "1248_HBL_PT_12_Fault" { S7_SetPoint := 'True'} : "stWinCCAlarm";
         "1249_HBL_PT_15_Fault" { S7_SetPoint := 'True'} : "stWinCCAlarm";
         "1251_HBL_PT_24_Fault" { S7_SetPoint := 'True'} : "stWinCCAlarm";
         "1252_HBL_TT_28_Fault" { S7_SetPoint := 'True'} : "stWinCCAlarm";
         "1253_HBL_TT_29_Fault" { S7_SetPoint := 'True'} : "stWinCCAlarm";
         "1254_HBL_TT_32_Fault" { S7_SetPoint := 'True'} : "stWinCCAlarm";
         "1255_HBL_CT_01_Fault" { S7_SetPoint := 'True'} : "stWinCCAlarm";
         "1256_HBL_CT_02_Fault" { S7_SetPoint := 'True'} : "stWinCCAlarm";
         "1258_HBL_TT_26_Fault" { S7_SetPoint := 'True'} : "stWinCCAlarm";
         "1259_HBL_TT_27_Fault" { S7_SetPoint := 'True'} : "stWinCCAlarm";
         "1260_HBL_FT_01_Fault" { S7_SetPoint := 'True'} : "stWinCCAlarm";
         "1262_HBL_TT_30_Fault" { S7_SetPoint := 'True'} : "stWinCCAlarm";
         "1263_HBL_TT_34_Fault" { S7_SetPoint := 'True'} : "stWinCCAlarm";
         "1264" { S7_SetPoint := 'True'} : "stWinCCAlarm";
         "1265" { S7_SetPoint := 'True'} : "stWinCCAlarm";
         "1266" { S7_SetPoint := 'True'} : "stWinCCAlarm";
         "1267" { S7_SetPoint := 'True'} : "stWinCCAlarm";
         "1268" { S7_SetPoint := 'True'} : "stWinCCAlarm";
         "1269" { S7_SetPoint := 'True'} : "stWinCCAlarm";
         "1270" { S7_SetPoint := 'True'} : "stWinCCAlarm";
         "1271" { S7_SetPoint := 'True'} : "stWinCCAlarm";
         "1272" { S7_SetPoint := 'True'} : "stWinCCAlarm";
         "1273" { S7_SetPoint := 'True'} : "stWinCCAlarm";
         "1274" { S7_SetPoint := 'True'} : "stWinCCAlarm";
         "1275" { S7_SetPoint := 'True'} : "stWinCCAlarm";
         "1276" { S7_SetPoint := 'True'} : "stWinCCAlarm";
         "1277" { S7_SetPoint := 'True'} : "stWinCCAlarm";
         "1278" { S7_SetPoint := 'True'} : "stWinCCAlarm";
         "1279" { S7_SetPoint := 'True'} : "stWinCCAlarm";
         "1280" { S7_SetPoint := 'True'} : "stWinCCAlarm";
         "1281" { S7_SetPoint := 'True'} : "stWinCCAlarm";
         "1282" { S7_SetPoint := 'True'} : "stWinCCAlarm";
         "1283" { S7_SetPoint := 'True'} : "stWinCCAlarm";
         "1284" { S7_SetPoint := 'True'} : "stWinCCAlarm";
         "1285" { S7_SetPoint := 'True'} : "stWinCCAlarm";
         "1286" { S7_SetPoint := 'True'} : "stWinCCAlarm";
         "1287" { S7_SetPoint := 'True'} : "stWinCCAlarm";
         "1288" { S7_SetPoint := 'True'} : "stWinCCAlarm";
         "1289" { S7_SetPoint := 'True'} : "stWinCCAlarm";
         "1290" { S7_SetPoint := 'True'} : "stWinCCAlarm";
         "1291" { S7_SetPoint := 'True'} : "stWinCCAlarm";
         "1292" { S7_SetPoint := 'True'} : "stWinCCAlarm";
         "1293" { S7_SetPoint := 'True'} : "stWinCCAlarm";
         "1294" { S7_SetPoint := 'True'} : "stWinCCAlarm";
         "1295" { S7_SetPoint := 'True'} : "stWinCCAlarm";
      END_STRUCT;
      "2-ProcessValues" : Struct
         "2018" : "stWinCCAlarm";
         "2028" { S7_SetPoint := 'True'} : "stWinCCAlarm";
         "2058" { S7_SetPoint := 'True'} : "stWinCCAlarm";
         "2100" { S7_SetPoint := 'True'} : "stWinCCAlarm";
         "2101" { S7_SetPoint := 'True'} : "stWinCCAlarm";
         "2102" { S7_SetPoint := 'True'} : "stWinCCAlarm";
         "2103" { S7_SetPoint := 'True'} : "stWinCCAlarm";
         "2105" { S7_SetPoint := 'True'} : "stWinCCAlarm";
         "2106" { S7_SetPoint := 'True'} : "stWinCCAlarm";
         "2107" : "stWinCCAlarm";
         "2108" { S7_SetPoint := 'True'} : "stWinCCAlarm";
         "2109" { S7_SetPoint := 'True'} : "stWinCCAlarm";
         "2110" { S7_SetPoint := 'True'} : "stWinCCAlarm";
         "2111" { S7_SetPoint := 'True'} : "stWinCCAlarm";
         "2112" { S7_SetPoint := 'True'} : "stWinCCAlarm";
         "2113" { S7_SetPoint := 'True'} : "stWinCCAlarm";
         "2114" { S7_SetPoint := 'True'} : "stWinCCAlarm";
         "2115" { S7_SetPoint := 'True'} : "stWinCCAlarm";
         "2116" { S7_SetPoint := 'True'} : "stWinCCAlarm";
         "2117" { S7_SetPoint := 'True'} : "stWinCCAlarm";
         "2301_HeatSourceTempDropCritical" { S7_SetPoint := 'True'} : "stWinCCAlarm";
         "2302_HeatSourceTempRiseCritical" { S7_SetPoint := 'True'} : "stWinCCAlarm";
         "2303_SuperheatCompressorHigh" { S7_SetPoint := 'True'} : "stWinCCAlarm";
         "2304_SuperheatCompressorLow" { S7_SetPoint := 'True'} : "stWinCCAlarm";
         "2305_OilFilterDeltaPHigh" { S7_SetPoint := 'True'} : "stWinCCAlarm";
         "2306_OilFilterDeltaPHighHigh" { S7_SetPoint := 'True'} : "stWinCCAlarm";
         "2307_EvaporatorDischargePressureMeanValue" { S7_SetPoint := 'True'} : "stWinCCAlarm";
         "2308_EvaporatorDischargePressureHigh" { S7_SetPoint := 'True'} : "stWinCCAlarm";
         "2309" { S7_SetPoint := 'True'} : "stWinCCAlarm";
      END_STRUCT;
      "3-Control" : Struct
         "3020" : "stWinCCAlarm";
         "3400_HydrolockProtectionActive" : "stWinCCAlarm";
         "3401_DripPanLevelHigh" { S7_SetPoint := 'True'} : "stWinCCAlarm";
      END_STRUCT;
      "4-Communication" : Struct
         dummy : Bool;
      END_STRUCT;
      "5-Auxiliaries" : Struct
         "5000_OilHeatingActivationFailure" : "stWinCCAlarm";
         "5001_OilHeatingDeactivationFailure" { S7_SetPoint := 'True'} : "stWinCCAlarm";
         "5200" : "stWinCCAlarm";
         "5201" { S7_SetPoint := 'True'} : "stWinCCAlarm";
         "5202" { S7_SetPoint := 'True'} : "stWinCCAlarm";
         "5203_CPC_SC_01_CommError" { S7_SetPoint := 'True'} : "stWinCCAlarm";
         "5204_CPC_SC_01_Tripped" { S7_SetPoint := 'True'} : "stWinCCAlarm";
         "5205" { S7_SetPoint := 'True'} : "stWinCCAlarm";
         "5206" { S7_SetPoint := 'True'} : "stWinCCAlarm";
         "5250_SSC_TT_01_Fault" { S7_SetPoint := 'True'} : "stWinCCAlarm";
         "5251_SSC_TT_02_Fault" { S7_SetPoint := 'True'} : "stWinCCAlarm";
         "5252_SSC_TT_03_Fault" { S7_SetPoint := 'True'} : "stWinCCAlarm";
         "5253_SSC_TT_04_Fault" { S7_SetPoint := 'True'} : "stWinCCAlarm";
         "5254_SSC_PIT_01_Fault" { S7_SetPoint := 'True'} : "stWinCCAlarm";
         "5255_SSC_PDT_01_Fault" { S7_SetPoint := 'True'} : "stWinCCAlarm";
         "5256_SSC_LT_01_Fault" { S7_SetPoint := 'True'} : "stWinCCAlarm";
         "5257_SSC_LT_01_Low" { S7_SetPoint := 'True'} : "stWinCCAlarm";
         "5258_SSC_PDT_01_High" { S7_SetPoint := 'True'} : "stWinCCAlarm";
         "5259_SSC_TT_02_High" { S7_SetPoint := 'True'} : "stWinCCAlarm";
         "5260_SSC_TT_03_Low" { S7_SetPoint := 'True'} : "stWinCCAlarm";
         "5261_SSC_PIT_01_Low" { S7_SetPoint := 'True'} : "stWinCCAlarm";
         "5262_DeltaT_ShaftSealHigh" : "stWinCCAlarm";
         "5263_SSC_PIT_01_High" { S7_SetPoint := 'True'} : "stWinCCAlarm";
         "5268_ShaftSealSystemShutdown" { S7_SetPoint := 'True'} : "stWinCCAlarm";
      END_STRUCT;
      "8-Events" : Struct
         "8000_State0_Initialize" : "stWinCCAlarm";
         "8001_State1_Offline" { S7_SetPoint := 'True'} : "stWinCCAlarm";
         "8002_State2_Standby" { S7_SetPoint := 'True'} : "stWinCCAlarm";
         "8003_State3_PrepareStart" { S7_SetPoint := 'True'} : "stWinCCAlarm";
         "8004_State4_Start" { S7_SetPoint := 'True'} : "stWinCCAlarm";
         "8005_State5_Warmup" { S7_SetPoint := 'True'} : "stWinCCAlarm";
         "8006_State6_Running" { S7_SetPoint := 'True'} : "stWinCCAlarm";
         "8007_State7_Stop" { S7_SetPoint := 'True'} : "stWinCCAlarm";
         "8010_Started" : "stWinCCAlarm";
         "8011_Stopped" { S7_SetPoint := 'True'} : "stWinCCAlarm";
         "8014_StartRequestHMI" { S7_SetPoint := 'True'} : "stWinCCAlarm";
         "8015_StartRequestApplication" { S7_SetPoint := 'True'} : "stWinCCAlarm";
         "8018_StopRequestHMI" { S7_SetPoint := 'True'} : "stWinCCAlarm";
         "8019_StopRequestApplication" { S7_SetPoint := 'True'} : "stWinCCAlarm";
         "8020_StopRequestCriticalAlarm" { S7_SetPoint := 'True'} : "stWinCCAlarm";
         "8021_StopRequestControllerFault" { S7_SetPoint := 'True'} : "stWinCCAlarm";
      END_STRUCT;
      "9-Diagnostics" : Struct
         "9021_CondenserBelowSinkTemp" : "stWinCCAlarm";
         "9022_CondensationAboveSinkTemp" { S7_SetPoint := 'True'} : "stWinCCAlarm";
         "9023" { S7_SetPoint := 'True'} : "stWinCCAlarm";
         "9024" { S7_SetPoint := 'True'} : "stWinCCAlarm";
         "9025" { S7_SetPoint := 'True'} : "stWinCCAlarm";
         "9026" { S7_SetPoint := 'True'} : "stWinCCAlarm";
         "9027" { S7_SetPoint := 'True'} : "stWinCCAlarm";
         "9028" { S7_SetPoint := 'True'} : "stWinCCAlarm";
         "9029" { S7_SetPoint := 'True'} : "stWinCCAlarm";
         "9030" { S7_SetPoint := 'True'} : "stWinCCAlarm";
         "9031" { S7_SetPoint := 'True'} : "stWinCCAlarm";
      END_STRUCT;
   END_VAR
BEGIN
END_DATA_BLOCK

ORGANIZATION_BLOCK "Main"   // OB1, FBD, ProgramCycle
TITLE = "Main Program Sweep (Cycle)"
{ S7_Optimized_Access := 'TRUE' }
VERSION : 0.1
// stored: AutoNumber true, IsIECCheckEnabled false, SetENOAutomatically false
   VAR_INPUT
      Initial_Call : Bool;   // Initial call of this OB
      Remanence : Bool;   // =True, if remanent data are available
   END_VAR
   VAR_TEMP
      dummy : Bool;
      InitError : Bool;
      RetVal10 : LReal;
   END_VAR
BEGIN

REGION Network 1: First cycle. Used for initialization
   // Use SET so that .bFirstCycle can be manually triggered
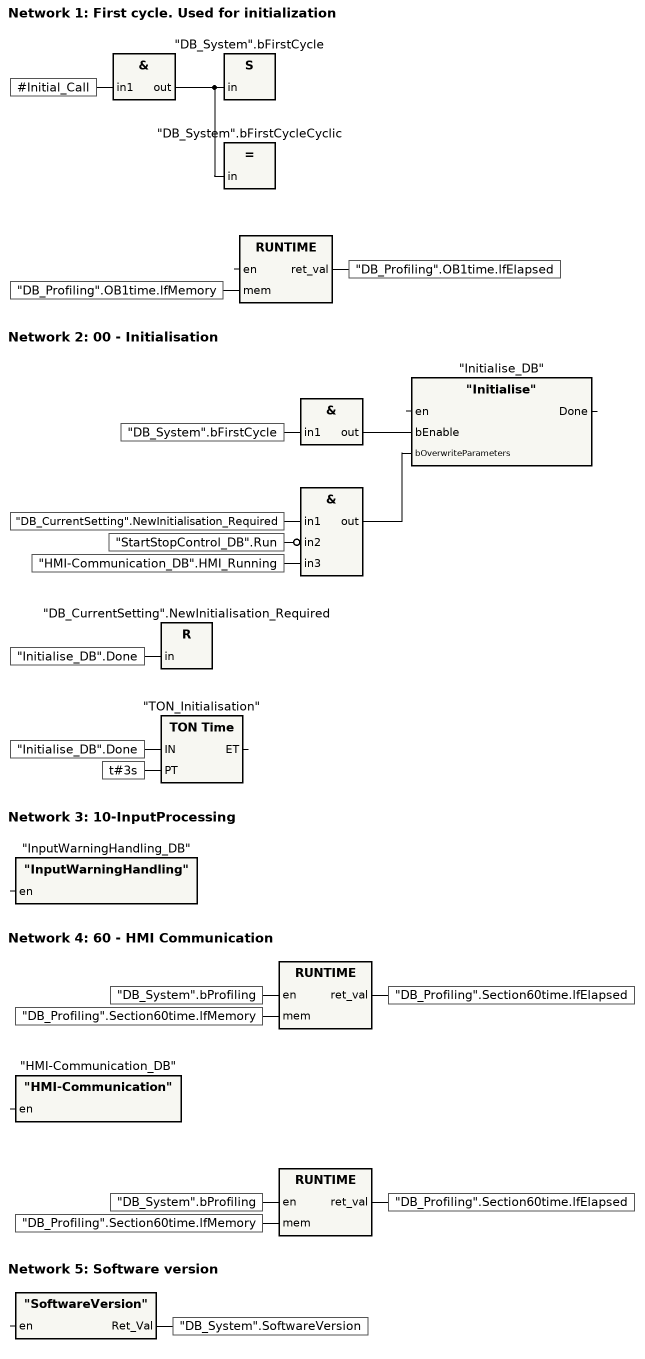
   // no SCL statement known for Runtime: written as a call
   IF #Initial_Call THEN "DB_System".bFirstCycle := TRUE; END_IF;
   "DB_System".bFirstCycleCyclic := #Initial_Call;
   "DB_Profiling".OB1time.lfElapsed := Runtime(mem := "DB_Profiling".OB1time.lfMemory);
END_REGION

REGION Network 2: 00 - Initialisation
   // Update alarm limits from DB_CurrentSettings on every restart
   // Load a new DB_CurrentSetting on NewInitialisation_Required, and update the alarm limits
   "Initialise_DB"(bEnable := "DB_System".bFirstCycle,   // "Initialise"
                   bOverwriteParameters := "DB_CurrentSetting".NewInitialisation_Required AND NOT "StartStopControl_DB".Run AND "HMI-Communication_DB".HMI_Running);
   IF "Initialise_DB".Done THEN "DB_CurrentSetting".NewInitialisation_Required := FALSE; END_IF;
   "TON_Initialisation".TON(IN := "Initialise_DB".Done, PT := t#3s);
END_REGION

REGION Network 3: 10-InputProcessing
   "InputWarningHandling_DB"();   // "InputWarningHandling"
END_REGION

REGION Network 4: 60 - HMI Communication
   // no SCL statement known for Runtime: written as a call
   IF "DB_System".bProfiling THEN
       "DB_Profiling".Section60time.lfElapsed := Runtime(mem := "DB_Profiling".Section60time.lfMemory);
   END_IF;
   "HMI-Communication_DB"();   // "HMI-Communication"
   IF "DB_System".bProfiling THEN
       "DB_Profiling".Section60time.lfElapsed := Runtime(mem := "DB_Profiling".Section60time.lfMemory);
   END_IF;
END_REGION

REGION Network 5: Software version
   "DB_System".SoftwareVersion := "SoftwareVersion"();
END_REGION

REGION Network 6: Reset first cycle
   // This network must be the last one in the program
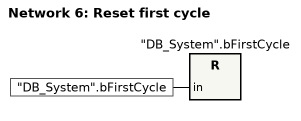
   IF "DB_System".bFirstCycle THEN "DB_System".bFirstCycle := FALSE; END_IF;
END_REGION
END_ORGANIZATION_BLOCK

FUNCTION_BLOCK "Initialise"   // FB25, FBD
{ S7_Optimized_Access := 'TRUE' }
AUTHOR : Heaten
VERSION : 0.1
// stored: AutoNumber true, IsIECCheckEnabled false, IsRetainMemResEnabled false, MemoryReserve 0, SetENOAutomatically false, UDAEnableTagReadback false
   VAR_INPUT
      bEnable { ExternalAccessible := 'False'; ExternalVisible := 'False'; ExternalWritable := 'False'} : Bool;
      bOverwriteParameters { ExternalAccessible := 'False'; ExternalVisible := 'False'; ExternalWritable := 'False'} : Bool;   // Overwrite DB_CurrentSetting from DB_StaticData
   END_VAR
   VAR_OUTPUT
      Done { ExternalAccessible := 'False'; ExternalVisible := 'False'; ExternalWritable := 'False'} : Bool;
   END_VAR
   VAR
      "Step" { ExternalAccessible := 'False'; ExternalVisible := 'False'; ExternalWritable := 'False'} : Int;
      Step_0 { ExternalAccessible := 'False'; ExternalVisible := 'False'; ExternalWritable := 'False'} : Bool;
      Step_1 { ExternalAccessible := 'False'; ExternalVisible := 'False'; ExternalWritable := 'False'} : Bool;
      Step_2 { ExternalAccessible := 'False'; ExternalVisible := 'False'; ExternalWritable := 'False'} : Bool;
      Step_3 { ExternalAccessible := 'False'; ExternalVisible := 'False'; ExternalWritable := 'False'} : Bool;
      Step_4 { ExternalAccessible := 'False'; ExternalVisible := 'False'; ExternalWritable := 'False'} : Bool;
      RetVal_Fluid { ExternalAccessible := 'False'; ExternalVisible := 'False'; ExternalWritable := 'False'} : Word;   // Static for debug purposes
      RetVal_System { ExternalAccessible := 'False'; ExternalVisible := 'False'; ExternalWritable := 'False'} : Word;   // Static for debug purposes
      RetVal_Compressor { ExternalAccessible := 'False'; ExternalVisible := 'False'; ExternalWritable := 'False'} : Word;   // Static for debug purposes
      A0003 { ExternalAccessible := 'False'; ExternalVisible := 'False'; ExternalWritable := 'False'} : "fbHMIEvent";
   END_VAR
   VAR_TEMP
      Busy : Bool;
   END_VAR
   VAR_TEMP   // added for the SCL form of the ladder/FBD networks
      _w1 : Bool;
   END_VAR
BEGIN

REGION Network 1 (SCL): Initialize step control
   IF (#bEnable = TRUE OR #bOverwriteParameters = TRUE) AND #Step_0 = FALSE AND #Step_1 = FALSE AND #Step_2 = FALSE AND #Step_3 = FALSE AND #Step_4 = FALSE THEN
       #Step_0 := TRUE;
       #Done := False;
   END_IF;
END_REGION

REGION Network 2 (SCL): Step_0: Set basic settings
   IF #Step_0 THEN

       "DB_State".State."0_Initialisation" := TRUE;

       "DB_State".State."1_Offline" :=
       "DB_State".State."2_Standby" :=
       "DB_State".State."3_PrepareStart" :=
       "DB_State".State."4_Start" :=
       "DB_State".State."5_Warmup" :=
       "DB_State".State."6_Running" :=
       "DB_State".State."7_Stop" := FALSE;

       //"DB_Alarms"."0001_WatchdogTimeoutOB1".bActive := FALSE;

       // Temporarily set some settings here. This should be changeable by the user via RETAIN variables.

      // "DB_CurrentSetting".VariableSetting.SystemType := 6;            // 1 = Test Station, 2 = Only cabinet, 3 = Ant, 4 = Bee, 5 = Cicada, 6 = HB-L4 Alpha
      // "DB_CurrentSetting".VariableSetting.FluidType := 1;             // 1 = R245fa
      // "DB_CurrentSetting".VariableSetting.CompressorType := 1;        // 1 = 1st Generation
      // "DB_CurrentSetting".VariableSetting.InstalledCompressors[8] := TRUE;
      "DB_CurrentSetting".VariableSetting.EnableViaHMI := TRUE;
       //"DB_Regulators".PerformanceControl.Settings.HeatSink.HeatSinkTemperatureControl_Active := TRUE;
       //"DB_Regulators".PerformanceControl.Settings.HeatSource.HeatSourceTemperatureControl_Active := FALSE;
       //"DB_Regulators".PerformanceControl.Settings.VariableControl.Control_Active := FALSE;

       //"DB_CurrentSetting".VariableSetting.ActiveCompressors := "DB_CurrentSetting".VariableSetting.InstalledCompressors;


       #Step_0 := FALSE;
       #Step_1 := TRUE;

   END_IF;
END_REGION

REGION Network 3 (SCL): Step_1: Currently not used

   IF #Step_1 THEN
       (* anything to do here? *)
       #Step_1 := FALSE;
       #Step_2 := TRUE;
   END_IF;
END_REGION

REGION Network 4: Step_2: Overwrite parameters
   // Load settings from Static DB if requested
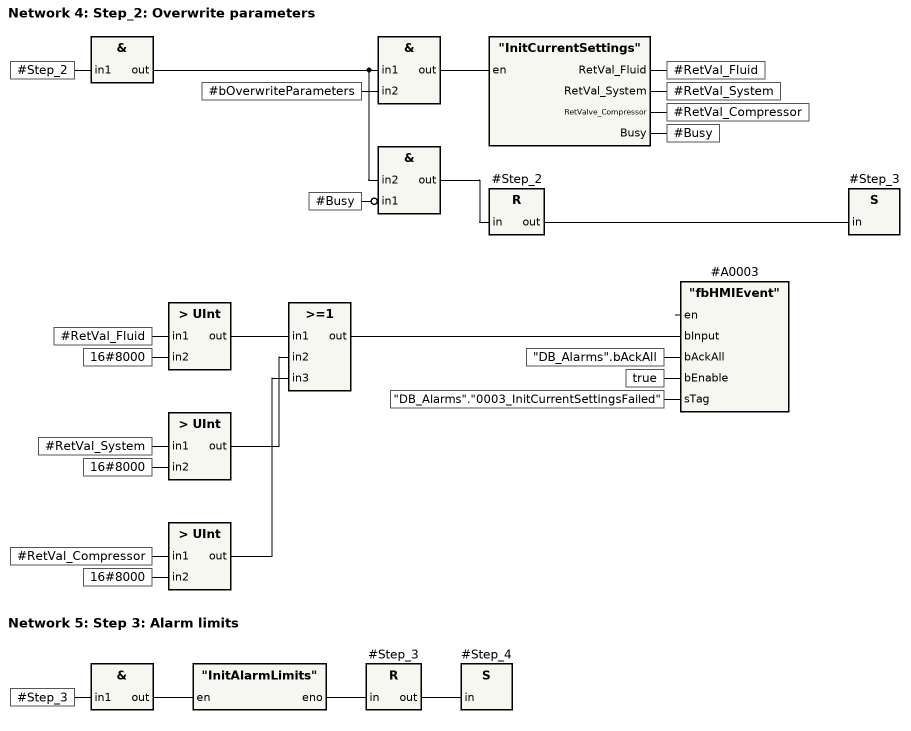
   IF #Step_2 AND #bOverwriteParameters THEN
       "InitCurrentSettings"(RetVal_Fluid => #RetVal_Fluid,
                             RetVal_System => #RetVal_System,
                             RetValve_Compressor => #RetVal_Compressor,
                             Busy => #Busy);
   END_IF;
   #_w1 := #Step_2 AND NOT #Busy;
   IF #_w1 THEN
       #Step_2 := FALSE;
       #Step_3 := TRUE;
   END_IF;
   #A0003(bInput := (#RetVal_Fluid > 16#8000) OR (#RetVal_System > 16#8000) OR (#RetVal_Compressor > 16#8000),   // "fbHMIEvent"
          bAckAll := "DB_Alarms".bAckAll,
          bEnable := true,
          sTag := "DB_Alarms"."0003_InitCurrentSettingsFailed");
END_REGION

REGION Network 5: Step 3: Alarm limits
   "InitAlarmLimits"(EN := #Step_3, ENO => #_w1);
   IF #_w1 THEN
       #Step_3 := FALSE;
       #Step_4 := TRUE;
   END_IF;
END_REGION

REGION Network 6 (SCL): Step 4
   IF #Step_4 THEN
       "DB_CurrentSetting".ParameterSet_Ordered := False;
       #Step_4 := FALSE;
       "DB_Alarms".bAckAll := TRUE; 
       #Done := True;
   END_IF;
END_REGION
END_FUNCTION_BLOCK

FUNCTION "InitCurrentSettings" : Void   // FC29, FBD
TITLE = Load data from DB_StaticData
{ S7_Optimized_Access := 'TRUE' }
AUTHOR : Heaten
VERSION : 0.1
// stored: AutoNumber true, IsIECCheckEnabled false, SetENOAutomatically false, UDAEnableTagReadback false
   VAR_OUTPUT
      RetVal_Fluid : Int;
      RetVal_System : Int;
      RetValve_Compressor : Int;
      Busy : Bool;
   END_VAR
   VAR_TEMP
      Busy_Fluid : Bool;
      Busy_System : Bool;
      Busy_Compressor : Bool;
      "Counter" : Int;
      Trigger : Bool;
   END_VAR
BEGIN

REGION Network 1: Load fluid data
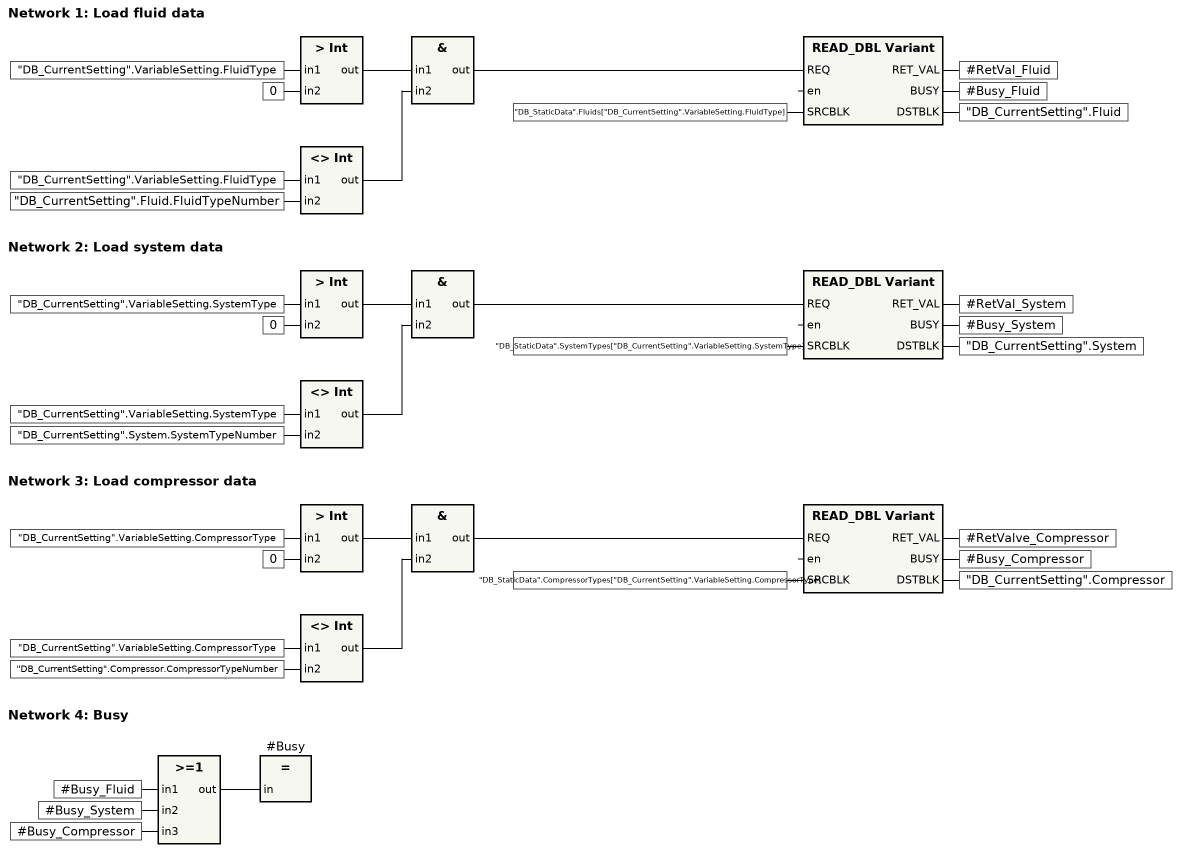
   #RetVal_Fluid := READ_DBL(REQ := ("DB_CurrentSetting".VariableSetting.FluidType > 0) AND ("DB_CurrentSetting".VariableSetting.FluidType <> "DB_CurrentSetting".Fluid.FluidTypeNumber),
                           SRCBLK := "DB_StaticData".Fluids["DB_CurrentSetting".VariableSetting.FluidType],
                           BUSY => #Busy_Fluid,
                           DSTBLK => "DB_CurrentSetting".Fluid);
END_REGION

REGION Network 2: Load system data
   #RetVal_System := READ_DBL(REQ := ("DB_CurrentSetting".VariableSetting.SystemType > 0) AND ("DB_CurrentSetting".VariableSetting.SystemType <> "DB_CurrentSetting".System.SystemTypeNumber),
                           SRCBLK := "DB_StaticData".SystemTypes["DB_CurrentSetting".VariableSetting.SystemType],
                           BUSY => #Busy_System,
                           DSTBLK => "DB_CurrentSetting".System);
END_REGION

REGION Network 3: Load compressor data
   #RetValve_Compressor := READ_DBL(REQ := ("DB_CurrentSetting".VariableSetting.CompressorType > 0) AND ("DB_CurrentSetting".VariableSetting.CompressorType <> "DB_CurrentSetting".Compressor.CompressorTypeNumber),
                           SRCBLK := "DB_StaticData".CompressorTypes["DB_CurrentSetting".VariableSetting.CompressorType],
                           BUSY => #Busy_Compressor,
                           DSTBLK => "DB_CurrentSetting".Compressor);
END_REGION

REGION Network 4: Busy
   #Busy := #Busy_Fluid OR #Busy_System OR #Busy_Compressor;
END_REGION
END_FUNCTION

FUNCTION_BLOCK "fbHMIEvent"   // FB39, FBD
{ S7_Optimized_Access := 'TRUE' }
VERSION : 0.1
// stored: AutoNumber true, IsIECCheckEnabled false, IsRetainMemResEnabled false, MemoryReserve 0, SetENOAutomatically false, UDAEnableTagReadback false
   VAR_INPUT
      bInput : Bool;
      bAckAll : Bool;
      bEnable : Bool;
   END_VAR
   VAR_IN_OUT
      sTag : "stEvent";
   END_VAR
   VAR
      Event : "fbEvent";
   END_VAR
BEGIN

REGION Network 1
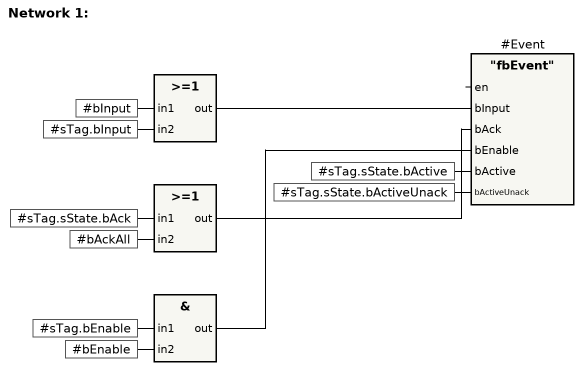
   #Event(bInput := #bInput OR #sTag.bInput,   // "fbEvent"
          bAck := #sTag.sState.bAck OR #bAckAll,
          bEnable := #sTag.bEnable AND #bEnable,
          bActive := #sTag.sState.bActive,
          bActiveUnack := #sTag.sState.bActiveUnack);
END_REGION
END_FUNCTION_BLOCK

FUNCTION_BLOCK "fbEvent"   // FB29, LAD
TITLE = Basic alarm
{ S7_Optimized_Access := 'TRUE' }
VERSION : 0.1
// stored: AutoNumber true, IsIECCheckEnabled false, IsRetainMemResEnabled false, MemoryReserve 0, SetENOAutomatically false, UDAEnableTagReadback false
   VAR_INPUT
      bInput : Bool;
      bAck : Bool;
      bEnable : Bool;
   END_VAR
   VAR_IN_OUT
      bActive : Bool;
      bActiveUnack : Bool;
   END_VAR
   VAR
      mActive : Bool;
   END_VAR
   VAR_TEMP   // added for the SCL form of the ladder/FBD networks
      _w1 : Bool;
   END_VAR
BEGIN

REGION Network 1: Alarm: reset if alarm is disabled or the alarm condition has cleared
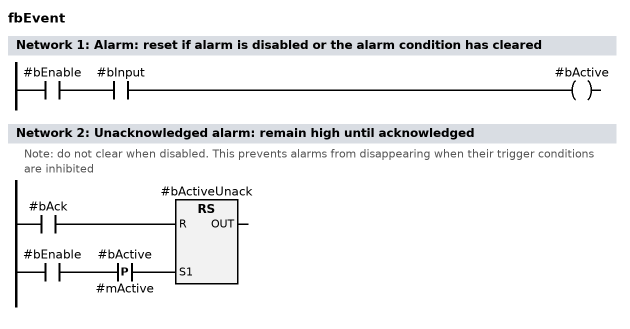
   RUNG wire#powerrail
      Contact( #bEnable )
      Contact( #bInput )
      Coil( #bActive )
   END_RUNG
   // the same network as SCL:
   #bActive := #bEnable AND #bInput;
END_REGION

REGION Network 2: Unacknowledged alarm: remain high until acknowledged
   // Note: do not clear when disabled. This prevents alarms from disappearing when their trigger conditions are inhibited
   RUNG wire#powerrail
      Contact( #bAck )
      S_RS(operand := #bActiveUnack, s1 := wire#w1)
   END_RUNG
   RUNG wire#powerrail
      Contact( #bEnable )
      P_Contact(operand := #bActive, bit := #mActive)
   END_RUNG wire#w1
   // the same network as SCL:
   #_w1 := #bEnable AND #bActive AND NOT #mActive;   // rising edge of #bActive
   #mActive := #bActive;
   IF #bAck THEN
       #bActiveUnack := FALSE;   // RS flip-flop
   END_IF;
   IF #_w1 THEN #bActiveUnack := TRUE; END_IF;
END_REGION
END_FUNCTION_BLOCK

FUNCTION "InitAlarmLimits" : Void   // FC6, FBD
TITLE = Alarm limits
{ S7_Optimized_Access := 'TRUE' }
AUTHOR : Heaten
VERSION : 0.1
// stored: AutoNumber true, IsIECCheckEnabled false, SetENOAutomatically false, UDAEnableTagReadback false
BEGIN

REGION Network 1 (SCL): 2018 Crankcase pressure HI
   // All alarms get .bEnabled on every restart to avoid accidental/forgotten alarm deactivation
   "DB_Alarms"."2018_HBL_PT_05_High".fLimit := "DB_CurrentSetting".Compressor.Limits.p_CrankCase_Max;
   "DB_Alarms"."2018_HBL_PT_05_High".bEnable := TRUE;
END_REGION

REGION Network 2 (SCL): 2028/2115 Oil pressure LO/LOLO
   // 2028 limit is dynamic, see FB19
   "DB_Alarms"."2028_HBL_PT_17_Low".bEnable := TRUE;

   // 2115 limit is dynamic, see FB19
   "DB_Alarms"."2115_HBL_PT_17_LowLow".bEnable := TRUE;
END_REGION

REGION Network 3 (SCL): 2058/2100 Crankcase oil sump temperature LO/HI
   // 2058 Low limit is dynamic based on crankcase condensing temperature, see FB19
   "DB_Alarms"."2058_HBL_TT_03_Low".bEnable := TRUE;

   "DB_Alarms"."2100_HBL_TT_03_High".fLimit := "DB_CurrentSetting".Fluid.Limits.T_OilTemperature_Critical;
   "DB_Alarms"."2100_HBL_TT_03_High".bEnable := TRUE;
END_REGION

REGION Network 4 (SCL): 2101 Heat sink suction temperature HI
   "DB_Alarms"."2101_HBL_TT_901_High".bEnable := TRUE;
   "DB_Alarms"."2101_HBL_TT_901_High".fLimit := "DB_CurrentSetting".MissingSetting.Misc.T_HeatSinkTemperatureIn_Max;
END_REGION

REGION Network 5 (SCL): 2102/2116 Compressor discharge pressure HI/HI HI
   // 100kPa below the HIHI limit (2116)
   // 100kPa below the HIHI limit
   "DB_Alarms"."2102_HBL_PT_503_High".fLimit := "DB_CurrentSetting".System.Limits.p_CompressorOut_Max - 100.0;
   "DB_Alarms"."2102_HBL_PT_503_High".bEnable := TRUE;

   "DB_Alarms"."2116_HBL_PT_503_HighHigh".bEnable := TRUE;
   "DB_Alarms"."2116_HBL_PT_503_HighHigh".fLimit := "DB_CurrentSetting".System.Limits.p_CompressorOut_Max;
END_REGION

REGION Network 6 (SCL): 2103 Heat sink discharge temperature HI
   "DB_Alarms"."2103_HBL_TT_518_High".fLimit := "DB_CurrentSetting".Fluid.Limits.T_HeatSinkTemperature_Max;
   "DB_Alarms"."2103_HBL_TT_518_High".bEnable := TRUE;
END_REGION

REGION Network 7 (SCL): 2105 Heat source suction temperature HI
   "DB_Alarms"."2105_HBL_TT_546_High".fLimit := "DB_CurrentSetting".Fluid.Limits.T_HeatSourceTemperature_Max;
   "DB_Alarms"."2105_HBL_TT_546_High".bEnable := TRUE;
END_REGION

REGION Network 8 (SCL): 2106 Control cabinet air temperature HI
   "DB_Alarms"."2106_HBL_TT_17_High".fLimit := "DB_CurrentSetting".StaticSetting.Limits.T_Cabinet_Max;
   "DB_Alarms"."2106_HBL_TT_17_High".bEnable := TRUE;
END_REGION

REGION Network 9 (SCL): 2107 Container air temperature HI
   "DB_Alarms"."2107_HBL_TT_16_High".fLimit := "DB_CurrentSetting".System.Limits.T_Housing_Max;
   "DB_Alarms"."2107_HBL_TT_16_High".bEnable := TRUE;
END_REGION

REGION Network 10 (SCL): 2108 Ambient air temperature HI
   "DB_Alarms"."2108_HBL_TT_18_High".fLimit := "DB_CurrentSetting".StaticSetting.Limits.T_Ambient_Max;
   "DB_Alarms"."2108_HBL_TT_18_High".bEnable := TRUE;
END_REGION

REGION Network 11 (SCL): 2109 Compressor motor temperature HI
   "DB_Alarms"."2109_HBL_TT_20_High".fLimit := "DB_CurrentSetting".Compressor.Limits.T_Motor_Max;
   "DB_Alarms"."2109_HBL_TT_20_High".bEnable := TRUE;
END_REGION

REGION Network 12 (SCL): 2110/2111 Oil sump wall temperature HI
   // Leave a temperature margin to avoid actually getting up into the critical temperature before triggering
   "DB_Alarms"."2110_HBL_TT_21_High".fLimit := "DB_CurrentSetting".Fluid.Limits.T_OilTemperature_Critical - 20.0;
   "DB_Alarms"."2110_HBL_TT_21_High".bEnable := TRUE;

   "DB_Alarms"."2111_HBL_TT_22_High".fLimit := "DB_CurrentSetting".Fluid.Limits.T_OilTemperature_Critical - 20.0;
   "DB_Alarms"."2111_HBL_TT_22_High".bEnable := TRUE;
END_REGION

REGION Network 13 (SCL): 2112 Oil separator oil level HI
   // ##FIX not in DB_CurrentSettings yet (or ever will be?)
   "DB_Alarms"."2112_HBL_LT_02_High".fLimit := 80.0;
   "DB_Alarms"."2112_HBL_LT_02_High".bEnable := TRUE;
END_REGION

REGION Network 14 (SCL): 2113/2114 Gas detectors HI
   // ##FIX not in DB_CurrentSettings yet
   "DB_Alarms"."2113_HBL_CT_01_High".fLimit := 1000.0;
   "DB_Alarms"."2113_HBL_CT_01_High".bEnable := TRUE;

   "DB_Alarms"."2114_HBL_CT_615_High".fLimit := 1000.0;
   "DB_Alarms"."2114_HBL_CT_615_High".bEnable := TRUE;
END_REGION

REGION Network 15 (SCL): 2301/2302 Heat source temperature rate of change
   // ##FIX not in DB_CurrentSettings yet
   "DB_Alarms"."2301_HeatSourceTempDropCritical".fLimit := -0.25;
   "DB_Alarms"."2301_HeatSourceTempDropCritical".bEnable := TRUE;

   "DB_Alarms"."2302_HeatSourceTempRiseCritical".fLimit := 0.25;
   "DB_Alarms"."2302_HeatSourceTempRiseCritical".bEnable := TRUE;
END_REGION

REGION Network 16 (SCL): 2303/2304 Superheat compressor suction HI/LO
   // ##FIX These limits are not in DB_CurrentSettings yet
   "DB_Alarms"."2303_SuperheatCompressor_High".fLimit := 30.0;
   "DB_Alarms"."2303_SuperheatCompressor_High".bEnable := TRUE;


   "DB_Alarms"."2304_SuperheatCompressor_Low".fLimit := "DB_CurrentSetting".System.Limits.T_SuperHeatCompressorIn_Min;
   "DB_Alarms"."2304_SuperheatCompressor_Low".bEnable := True;
END_REGION

REGION Network 17 (SCL): 2305/2306 Oil filter delta P HI/HIHI
   "DB_Alarms"."2305_OilFilterDeltaP_High".fLimit := "DB_CurrentSetting".MissingSetting.Compressor.OilFilterDeltaPWarning;
   "DB_Alarms"."2305_OilFilterDeltaP_High".bEnable := TRUE;

   "DB_Alarms"."2306_OilFilterDeltaP_HighHigh".fLimit := "DB_CurrentSetting".MissingSetting.Compressor.OilFilterDeltaPCritical;
   "DB_Alarms"."2306_OilFilterDeltaP_HighHigh".bEnable := TRUE;
END_REGION

REGION Network 18 (SCL): 2308 Evaporator discharge pressure HI
   "DB_Alarms"."2308_EvaporatorDischargePressureHigh".fLimit := "DB_CurrentSetting".System.Limits.p_EvaporatorOut_Max;
   "DB_Alarms"."2308_EvaporatorDischargePressureHigh".bEnable := TRUE;
END_REGION

REGION Network 19 (SCL): 5205 CPC tank level HI
   "DB_Alarms"."5205_CPC_LT_870_High".fLimit := 90.0;
   "DB_Alarms"."5205_CPC_LT_870_High".bEnable := TRUE;
END_REGION

REGION Network 20 (SCL): 5257 SSC barrier reservoir LO
   "DB_Alarms"."5257_SSC_LT_01_Low".fLimit := 5.0;
   "DB_Alarms"."5257_SSC_LT_01_Low".bEnable := TRUE;
END_REGION

REGION Network 21 (SCL): 5258 SSC barrier fluid pump differential pressure HI
   "DB_Alarms"."5258_SSC_PDT_01_High".fLimit := 200.0;
   "DB_Alarms"."5258_SSC_PDT_01_High".bEnable := TRUE;
END_REGION

REGION Network 22 (SCL): 5259 SSC seal discharge temperature HI
   "DB_Alarms"."5259_SSC_TT_02_High".fLimit := 110.0;
   "DB_Alarms"."5259_SSC_TT_02_High".bEnable := TRUE;
END_REGION

REGION Network 23 (SCL): 5260 SSC circulation pump suction temperature LO
   "DB_Alarms"."5260_SSC_TT_03_Low".fLimit := 10.0;
   "DB_Alarms"."5260_SSC_TT_03_Low".bEnable := TRUE;
END_REGION

